  MoveC 7172 to (-6.47, 57.05, -11) mm, rotated rx -180 ry 0 rz 90 deg; joints [75.622, -17.705, 85.85, 0, 21.855, 75.622] to (-5.97, 56.82, -11) mm, rotated rx 180 ry 0 rz 90 deg; joints [75.618, -17.695, 85.811, 0, 21.884, 75.618]
  MoveC 7173 to (11.96, 58.42, -11) mm, rotated rx 180 ry 0 rz 90 deg; joints [75.821, -17.382, 84.57, 0, 22.812, 75.821] to (29.85, 60.38, -11) mm, rotated rx -180 ry 0 rz 90 deg; joints [76.031, -17.055, 83.319, 0, 23.736, 76.031]
  MoveC 7174 to (37.63, 61.41, -11) mm, rotated rx 180 ry 0 rz 90 deg; joints [76.126, -16.91, 82.773, 0, 24.137, 76.126] to (45.39, 62.55, -11) mm, rotated rx -180 ry 0 rz 90 deg; joints [76.225, -16.762, 82.226, 0, 24.537, 76.225]
  MoveL 7175 to (45.39, 69.07, -11) mm, rotated rx 180 ry 0 rz 90 deg; joints [76.435, -16.794, 82.342, 0, 24.452, 76.435]
  MoveC 7176 to (32.64, 69.9, -11) mm, rotated rx 180 ry 0 rz 90 deg; joints [76.362, -17.047, 83.287, 0, 23.76, 76.362] to (19.88, 70.48, -11) mm, rotated rx -180 ry 0 rz 90 deg; joints [76.279, -17.291, 84.218, 0, 23.073, 76.279]
  MoveC 7177 to (17, 70.58, -11) mm, rotated rx 180 ry 0 rz 90 deg; joints [76.26, -17.344, 84.426, 0, 22.919, 76.26] to (14.12, 70.67, -11) mm, rotated rx 180 ry 0 rz 90 deg; joints [76.24, -17.398, 84.633, 0, 22.765, 76.24]
  MoveL 7178 to (13.87, 63.13, -11) mm, rotated rx -180 ry 0 rz 90 deg; joints [75.991, -17.368, 84.518, 0, 22.85, 75.991]
  MoveL 7179 to (13.87, 63.13, -8) mm, rotated rx 180 ry 0 rz 90 deg; joints [75.991, -17.522, 84.62, 0, 22.902, 75.991]
  Establecer velocidad (1000.0 mm/s)
  MoveL 7180 to (13.87, 63.13, 10) mm, rotated rx 180 ry 0 rz 90 deg; joints [75.991, -18.443, 85.222, 0, 23.22, 75.991]
  Establecer velocidad (66.7 mm/s)
  MoveL 7181 to (-0.84, 59.62, 10) mm, rotated rx 180 ry 0 rz 90 deg; joints [75.754, -18.697, 86.204, 0, 22.493, 75.754]
  MoveL 7182 to (-0.84, 59.62, -8) mm, rotated rx -180 ry 0 rz 90 deg; joints [75.754, -17.772, 85.602, 0, 22.17, 75.754]
  MoveL 7183 to (0.35, 58.68, -8.41) mm, rotated rx -180 ry 0 rz 90 deg; joints [75.733, -17.725, 85.487, 0, 22.239, 75.733]
  MoveL 7184 to (1.74, 58.06, -8.81) mm, rotated rx 180 ry 0 rz 90 deg; joints [75.724, -17.677, 85.364, 0, 22.313, 75.724]
  MoveL 7185 to (3.23, 57.78, -9.22) mm, rotated rx -180 ry 0 rz 90 deg; joints [75.727, -17.628, 85.239, 0, 22.389, 75.727]
  MoveL 7186 to (4.75, 57.85, -9.62) mm, rotated rx -180 ry 0 rz 90 deg; joints [75.742, -17.58, 85.119, 0, 22.461, 75.742]
  MoveL 7187 to (6.21, 58.28, -10.03) mm, rotated rx 180 ry 0 rz 90 deg; joints [75.769, -17.535, 85.009, 0, 22.526, 75.769]
  MoveL 7188 to (7.53, 59.03, -10.44) mm, rotated rx 180 ry 0 rz 90 deg; joints [75.804, -17.494, 84.915, 0, 22.579, 75.804]
  MoveL 7189 to (8.65, 60.06, -10.84) mm, rotated rx 180 ry 0 rz 90 deg; joints [75.847, -17.458, 84.841, 0, 22.617, 75.847]
  MoveL 7190 to (9.46, 61.34, -11.25) mm, rotated rx 180 ry 0 rz 90 deg; joints [75.896, -17.428, 84.792, 0, 22.636, 75.896]
  MoveL 7191 to (14.11, 70.46, -11.25) mm, rotated rx 180 ry 0 rz 90 deg; joints [76.233, -17.384, 84.621, 0, 22.763, 76.233]
  MoveL 7192 to (7.11, 70.69, -11.25) mm, rotated rx 180 ry 0 rz 90 deg; joints [76.184, -17.512, 85.124, 0, 22.388, 76.184]
  MoveL 7193 to (-16.58, 71.34, -11.25) mm, rotated rx -180 ry 0 rz 90 deg; joints [76.011, -17.928, 86.802, 0, 21.125, 76.011]
  MoveC 7194 to (-18.77, 68.61, -11.25) mm, rotated rx 180 ry 0 rz 90 deg; joints [75.902, -17.953, 86.907, 0, 21.046, 75.902] to (-18.5, 65.12, -11.25) mm, rotated rx -180 ry 0 rz 90 deg; joints [75.788, -17.933, 86.827, 0, 21.107, 75.788]
  MoveL 7195 to (-8.05, 58.36, -11.25) mm, rotated rx 180 ry 0 rz 90 deg; joints [75.652, -17.726, 85.977, 0, 21.749, 75.652]
  MoveL 7196 to (-6.15, 57.11, -11.25) mm, rotated rx 180 ry 0 rz 90 deg; joints [75.626, -17.687, 85.82, 0, 21.867, 75.626]
  MoveC 7197 to (-5.87, 56.99, -11.25) mm, rotated rx -180 ry 0 rz 90 deg; joints [75.625, -17.681, 85.798, 0, 21.883, 75.625] to (-5.57, 56.96, -11.25) mm, rotated rx -180 ry 0 rz 90 deg; joints [75.627, -17.676, 85.777, 0, 21.899, 75.627]
  MoveC 7198 to (11.68, 58.54, -11.25) mm, rotated rx -180 ry 0 rz 90 deg; joints [75.823, -17.374, 84.583, 0, 22.791, 75.823] to (28.9, 60.45, -11.25) mm, rotated rx 180 ry 0 rz 90 deg; joints [76.025, -17.061, 83.381, 0, 23.681, 76.025]
  MoveL 7199 to (40.27, 62.01, -11.25) mm, rotated rx -180 ry 0 rz 90 deg; joints [76.167, -16.848, 82.582, 0, 24.266, 76.167]
  MoveL 7200 to (42.53, 62.35, -11.25) mm, rotated rx -180 ry 0 rz 90 deg; joints [76.196, -16.805, 82.423, 0, 24.382, 76.196]
  MoveL 7201 to (42.53, 69.03, -11.25) mm, rotated rx 180 ry 0 rz 90 deg; joints [76.411, -16.838, 82.542, 0, 24.295, 76.411]
  MoveC 7202 to (29.09, 69.85, -11.25) mm, rotated rx 180 ry 0 rz 90 deg; joints [76.332, -17.102, 83.534, 0, 23.567, 76.332] to (15.63, 70.41, -11.25) mm, rotated rx 180 ry 0 rz 90 deg; joints [76.243, -17.356, 84.512, 0, 22.844, 76.243]
  MoveL 7203 to (14.11, 70.46, -11.25) mm, rotated rx 180 ry 0 rz 90 deg; joints [76.233, -17.384, 84.621, 0, 22.763, 76.233]
  MoveL 7204 to (13.87, 62.91, -11.25) mm, rotated rx 180 ry 0 rz 90 deg; joints [75.984, -17.354, 84.506, 0, 22.849, 75.984]
  MoveL 7205 to (13.87, 62.91, -8.25) mm, rotated rx 180 ry 0 rz 90 deg; joints [75.984, -17.508, 84.608, 0, 22.9, 75.984]
  Establecer velocidad (1000.0 mm/s)
  MoveL 7206 to (13.87, 62.91, 10) mm, rotated rx -180 ry 0 rz 90 deg; joints [75.984, -18.442, 85.219, 0, 23.223, 75.984]
  Establecer velocidad (66.7 mm/s)
  MoveL 7207 to (34.75, 17.39, 10) mm, rotated rx 180 ry 0 rz 90 deg; joints [74.689, -17.806, 82.854, 0, 24.952, 74.689]
  MoveL 7208 to (34.75, 17.39, -8) mm, rotated rx 180 ry 0 rz 90 deg; joints [74.689, -16.893, 82.249, 0, 24.644, 74.689]
  MoveL 7209 to (34.95, 18.89, -8.41) mm, rotated rx 180 ry 0 rz 90 deg; joints [74.738, -16.877, 82.251, 0, 24.626, 74.738]
  MoveL 7210 to (34.77, 20.4, -8.81) mm, rotated rx -180 ry 0 rz 90 deg; joints [74.785, -16.868, 82.28, 0, 24.588, 74.785]
  MoveL 7211 to (34.27, 21.84, -9.22) mm, rotated rx 180 ry 0 rz 90 deg; joints [74.827, -16.865, 82.332, 0, 24.534, 74.827]
  MoveL 7212 to (33.46, 23.12, -9.62) mm, rotated rx -180 ry 0 rz 90 deg; joints [74.861, -16.867, 82.402, 0, 24.465, 74.861]
  MoveL 7213 to (32.38, 24.2, -10.03) mm, rotated rx 180 ry 0 rz 90 deg; joints [74.886, -16.874, 82.488, 0, 24.386, 74.886]
  MoveL 7214 to (31.1, 25.01, -10.44) mm, rotated rx -180 ry 0 rz 90 deg; joints [74.901, -16.882, 82.583, 0, 24.299, 74.901]
  MoveL 7215 to (29.66, 25.51, -10.84) mm, rotated rx 180 ry 0 rz 90 deg; joints [74.904, -16.892, 82.683, 0, 24.209, 74.904]
  MoveL 7216 to (28.15, 25.66, -11.25) mm, rotated rx -180 ry 0 rz 90 deg; joints [74.896, -16.902, 82.781, 0, 24.12, 74.896]
  MoveC 7217 to (21.42, 25.67, -11.25) mm, rotated rx 180 ry 0 rz 90 deg; joints [74.838, -17.031, 83.268, 0, 23.763, 74.838] to (14.69, 25.64, -11.25) mm, rotated rx 180 ry 0 rz 90 deg; joints [74.778, -17.159, 83.751, 0, 23.408, 74.778]
  MoveL 7218 to (13.74, 25.57, -11.25) mm, rotated rx 180 ry 0 rz 90 deg; joints [74.767, -17.176, 83.818, 0, 23.358, 74.767]
  MoveC 7219 to (11.74, 24.17, -11.25) mm, rotated rx 180 ry 0 rz 90 deg; joints [74.704, -17.206, 83.934, 0, 23.273, 74.704] to (11.18, 21.8, -11.25) mm, rotated rx 180 ry 0 rz 90 deg; joints [74.622, -17.205, 83.927, 0, 23.277, 74.622]
  MoveL 7220 to (11.34, 21.32, -11.25) mm, rotated rx 180 ry 0 rz 90 deg; joints [74.609, -17.199, 83.906, 0, 23.293, 74.609]
  MoveL 7221 to (14.96, 11.54, -11.25) mm, rotated rx 180 ry 0 rz 90 deg; joints [74.325, -17.08, 83.453, 0, 23.628, 74.325]
  MoveC 7222 to (15.41, 10.71, -11.25) mm, rotated rx 180 ry 0 rz 90 deg; joints [74.303, -17.067, 83.403, 0, 23.664, 74.303] to (16.08, 10.04, -11.25) mm, rotated rx 180 ry 0 rz 90 deg; joints [74.287, -17.051, 83.342, 0, 23.709, 74.287]
  MoveL 7223 to (27.98, 1.22, -11.25) mm, rotated rx -180 ry 0 rz 90 deg; joints [74.113, -16.773, 82.303, 0, 24.47, 74.113]
  MoveC 7224 to (28.43, 0.91, -11.25) mm, rotated rx 180 ry 0 rz 90 deg; joints [74.107, -16.762, 82.264, 0, 24.498, 74.107] to (28.9, 0.64, -11.25) mm, rotated rx -180 ry 0 rz 90 deg; joints [74.102, -16.751, 82.224, 0, 24.528, 74.102]
  MoveC 7225 to (31.23, 0.68, -11.25) mm, rotated rx 180 ry 0 rz 90 deg; joints [74.125, -16.706, 82.055, 0, 24.65, 74.125] to (33.09, 2.08, -11.25) mm, rotated rx 180 ry 0 rz 90 deg; joints [74.186, -16.677, 81.949, 0, 24.728, 74.186]
  MoveL 7226 to (33.64, 2.87, -11.25) mm, rotated rx 180 ry 0 rz 90 deg; joints [74.216, -16.67, 81.925, 0, 24.745, 74.216]
  MoveL 7227 to (42.53, 15.9, -11.25) mm, rotated rx 180 ry 0 rz 90 deg; joints [74.709, -16.565, 81.54, 0, 25.025, 74.709]
  MoveL 7228 to (42.53, 25.35, -11.25) mm, rotated rx -180 ry 0 rz 90 deg; joints [75.01, -16.616, 81.727, 0, 24.889, 75.01]
  MoveL 7229 to (42.3, 25.48, -11.25) mm, rotated rx -180 ry 0 rz 90 deg; joints [75.012, -16.621, 81.747, 0, 24.875, 75.012]
  MoveL 7230 to (41.22, 25.52, -11.25) mm, rotated rx 180 ry 0 rz 90 deg; joints [75.004, -16.643, 81.827, 0, 24.817, 75.004]
  MoveC 7231 to (34.69, 25.61, -11.25) mm, rotated rx -180 ry 0 rz 90 deg; joints [74.951, -16.774, 82.306, 0, 24.468, 74.951] to (28.15, 25.66, -11.25) mm, rotated rx -180 ry 0 rz 90 deg; joints [74.896, -16.902, 82.781, 0, 24.12, 74.896]
  MoveL 7232 to (28.12, 18.11, -11.25) mm, rotated rx -180 ry 0 rz 90 deg; joints [74.654, -16.863, 82.635, 0, 24.228, 74.654]
  MoveL 7233 to (28.12, 18.11, -8.25) mm, rotated rx -180 ry 0 rz 90 deg; joints [74.654, -17.015, 82.737, 0, 24.278, 74.654]
  Establecer velocidad (1000.0 mm/s)
  MoveL 7234 to (28.12, 18.11, 10) mm, rotated rx 180 ry 0 rz 90 deg; joints [74.654, -17.942, 83.35, 0, 24.592, 74.654]
  Establecer velocidad (66.7 mm/s)
  MoveL 7235 to (14.48, -62.46, 10) mm, rotated rx 180 ry 0 rz 90 deg; joints [71.966, -17.733, 82.59, 0, 25.143, 71.966]
  MoveL 7236 to (14.48, -62.46, -8) mm, rotated rx -180 ry 0 rz 90 deg; joints [71.966, -16.821, 81.985, 0, 24.836, 71.966]
  MoveL 7237 to (14.35, -63.97, -8.41) mm, rotated rx 180 ry 0 rz 90 deg; joints [71.918, -16.793, 81.945, 0, 24.848, 71.918]
  MoveL 7238 to (14.59, -65.48, -8.81) mm, rotated rx 180 ry 0 rz 90 deg; joints [71.873, -16.758, 81.878, 0, 24.88, 71.873]
  MoveL 7239 to (15.16, -66.89, -9.22) mm, rotated rx 180 ry 0 rz 90 deg; joints [71.835, -16.717, 81.79, 0, 24.927, 71.835]
  MoveL 7240 to (16.03, -68.13, -9.62) mm, rotated rx -180 ry 0 rz 90 deg; joints [71.804, -16.671, 81.684, 0, 24.987, 71.804]
  MoveL 7241 to (17.15, -69.16, -10.03) mm, rotated rx 180 ry 0 rz 90 deg; joints [71.784, -16.622, 81.565, 0, 25.057, 71.784]
  MoveL 7242 to (18.47, -69.91, -10.44) mm, rotated rx 180 ry 0 rz 90 deg; joints [71.774, -16.57, 81.438, 0, 25.132, 71.774]
  MoveL 7243 to (19.92, -70.36, -10.84) mm, rotated rx 180 ry 0 rz 90 deg; joints [71.775, -16.517, 81.308, 0, 25.209, 71.775]
  MoveL 7244 to (21.44, -70.43, -11.25) mm, rotated rx 180 ry 0 rz 90 deg; joints [71.788, -16.466, 81.182, 0, 25.284, 71.788]
  MoveC 7245 to (30.97, -70.02, -11.25) mm, rotated rx 180 ry 0 rz 90 deg; joints [71.898, -16.275, 80.498, 0, 25.777, 71.898] to (40.49, -69.51, -11.25) mm, rotated rx -180 ry 0 rz 90 deg; joints [72.01, -16.08, 79.81, 0, 26.27, 72.01]
  MoveC 7246 to (41.74, -68.34, -11.25) mm, rotated rx -180 ry 0 rz 90 deg; joints [72.059, -16.062, 79.746, 0, 26.316, 72.059] to (42.53, -66.81, -11.25) mm, rotated rx -180 ry 0 rz 90 deg; joints [72.114, -16.055, 79.723, 0, 26.332, 72.114]
  MoveL 7247 to (42.53, -62.79, -11.25) mm, rotated rx -180 ry 0 rz 90 deg; joints [72.239, -16.082, 79.819, 0, 26.263, 72.239]
  MoveC 7248 to (32.93, -50.94, -11.25) mm, rotated rx 180 ry 0 rz 90 deg; joints [72.513, -16.36, 80.802, 0, 25.558, 72.513] to (23.22, -39.19, -11.25) mm, rotated rx -180 ry 0 rz 90 deg; joints [72.786, -16.63, 81.777, 0, 24.853, 72.786]
  MoveL 7249 to (22.31, -38.38, -11.25) mm, rotated rx 180 ry 0 rz 90 deg; joints [72.803, -16.653, 81.861, 0, 24.792, 72.803]
  MoveL 7250 to (13.74, -31.32, -11.25) mm, rotated rx 180 ry 0 rz 90 deg; joints [72.943, -16.863, 82.636, 0, 24.227, 72.943]
  MoveC 7251 to (11.26, -30.82, -11.25) mm, rotated rx 180 ry 0 rz 90 deg; joints [72.935, -16.914, 82.826, 0, 24.088, 72.935] to (9, -31.97, -11.25) mm, rotated rx 180 ry 0 rz 90 deg; joints [72.876, -16.95, 82.962, 0, 23.988, 72.876]
  MoveC 7252 to (8.77, -32.34, -11.25) mm, rotated rx -180 ry 0 rz 90 deg; joints [72.862, -16.952, 82.971, 0, 23.982, 72.862] to (8.61, -32.74, -11.25) mm, rotated rx -180 ry 0 rz 90 deg; joints [72.848, -16.953, 82.973, 0, 23.98, 72.848]
  MoveL 7253 to (-0.76, -67.29, -11.25) mm, rotated rx 180 ry 0 rz 90 deg; joints [71.657, -16.921, 82.853, 0, 24.068, 71.657]
  MoveC 7254 to (-0.84, -67.76, -11.25) mm, rotated rx -180 ry 0 rz 90 deg; joints [71.641, -16.919, 82.847, 0, 24.072, 71.641] to (-0.81, -68.23, -11.25) mm, rotated rx 180 ry 0 rz 90 deg; joints [71.626, -16.916, 82.833, 0, 24.082, 71.626]
  MoveC 7255 to (0.29, -70.18, -11.25) mm, rotated rx 180 ry 0 rz 90 deg; joints [71.576, -16.882, 82.709, 0, 24.173, 71.576] to (2.37, -71.02, -11.25) mm, rotated rx -180 ry 0 rz 90 deg; joints [71.572, -16.837, 82.541, 0, 24.296, 71.572]
  MoveC 7256 to (11.91, -70.77, -11.25) mm, rotated rx -180 ry 0 rz 90 deg; joints [71.679, -16.653, 81.863, 0, 24.79, 71.679] to (21.44, -70.43, -11.25) mm, rotated rx 180 ry 0 rz 90 deg; joints [71.788, -16.466, 81.182, 0, 25.284, 71.788]
  MoveL 7257 to (21.14, -62.89, -11.25) mm, rotated rx 180 ry 0 rz 90 deg; joints [72.021, -16.521, 81.383, 0, 25.138, 72.021]
  MoveL 7258 to (21.14, -62.89, -8.25) mm, rotated rx 180 ry 0 rz 90 deg; joints [72.021, -16.673, 81.485, 0, 25.188, 72.021]
  Establecer velocidad (1000.0 mm/s)
  MoveL 7259 to (21.14, -62.89, 10) mm, rotated rx 180 ry 0 rz 90 deg; joints [72.021, -17.596, 82.099, 0, 25.497, 72.021]
  Establecer velocidad (66.7 mm/s)
  MoveL 7260 to (-37.75, -51.92, 10) mm, rotated rx 180 ry 0 rz 90 deg; joints [71.757, -18.775, 86.512, 0, 22.263, 71.757]
  MoveL 7261 to (-37.75, -51.92, -8) mm, rotated rx 180 ry 0 rz 90 deg; joints [71.757, -17.849, 85.91, 0, 21.939, 71.757]
  MoveL 7262 to (-36.33, -52.48, -8.41) mm, rotated rx -180 ry 0 rz 90 deg; joints [71.754, -17.801, 85.786, 0, 22.015, 71.754]
  MoveL 7263 to (-34.83, -52.68, -8.81) mm, rotated rx 180 ry 0 rz 90 deg; joints [71.764, -17.753, 85.664, 0, 22.089, 71.764]
  MoveL 7264 to (-33.31, -52.54, -9.22) mm, rotated rx 180 ry 0 rz 90 deg; joints [71.784, -17.706, 85.548, 0, 22.158, 71.784]
  MoveL 7265 to (-31.87, -52.07, -9.62) mm, rotated rx 180 ry 0 rz 90 deg; joints [71.815, -17.663, 85.445, 0, 22.218, 71.815]
  MoveL 7266 to (-30.56, -51.29, -10.03) mm, rotated rx -180 ry 0 rz 90 deg; joints [71.854, -17.624, 85.358, 0, 22.265, 71.854]
  MoveL 7267 to (-29.46, -50.25, -10.44) mm, rotated rx 180 ry 0 rz 90 deg; joints [71.899, -17.589, 85.292, 0, 22.297, 71.899]
  MoveL 7268 to (-28.62, -48.98, -10.84) mm, rotated rx 180 ry 0 rz 90 deg; joints [71.949, -17.561, 85.248, 0, 22.313, 71.949]
  MoveL 7269 to (-28.11, -47.55, -11.25) mm, rotated rx -180 ry 0 rz 90 deg; joints [72, -17.539, 85.231, 0, 22.308, 72]
  MoveL 7270 to (-22.44, -25.59, -11.25) mm, rotated rx 180 ry 0 rz 90 deg; joints [72.769, -17.562, 85.322, 0, 22.24, 72.769]
  MoveC 7271 to (-22.4, -25.35, -11.25) mm, rotated rx 180 ry 0 rz 90 deg; joints [72.777, -17.563, 85.324, 0, 22.238, 72.777] to (-22.41, -25.11, -11.25) mm, rotated rx 180 ry 0 rz 90 deg; joints [72.784, -17.564, 85.33, 0, 22.234, 72.784]
  MoveC 7272 to (-23.45, -22.93, -11.25) mm, rotated rx 180 ry 0 rz 90 deg; joints [72.845, -17.594, 85.45, 0, 22.145, 72.845] to (-25.59, -21.78, -11.25) mm, rotated rx -180 ry 0 rz 90 deg; joints [72.861, -17.638, 85.623, 0, 22.015, 72.861]
  MoveL 7273 to (-26.06, -21.85, -11.25) mm, rotated rx -180 ry 0 rz 90 deg; joints [72.854, -17.646, 85.654, 0, 21.991, 72.854]
  MoveL 7274 to (-33.64, -23.38, -11.25) mm, rotated rx -180 ry 0 rz 90 deg; joints [72.727, -17.768, 86.147, 0, 21.621, 72.727]
  MoveL 7275 to (-63.02, -29.41, -11.25) mm, rotated rx 180 ry 0 rz 90 deg; joints [72.225, -18.217, 88.022, 0, 20.195, 72.225]
  MoveL 7276 to (-70.18, -30.91, -11.25) mm, rotated rx 180 ry 0 rz 90 deg; joints [72.099, -18.321, 88.472, 0, 19.849, 72.099]
  MoveC 7277 to (-71.74, -31.8, -11.25) mm, rotated rx 180 ry 0 rz 90 deg; joints [72.052, -18.341, 88.557, 0, 19.783, 72.052] to (-72.48, -33.43, -11.25) mm, rotated rx -180 ry 0 rz 90 deg; joints [71.99, -18.344, 88.572, 0, 19.772, 71.99]
  MoveL 7278 to (-72.5, -33.64, -11.25) mm, rotated rx 180 ry 0 rz 90 deg; joints [71.983, -18.343, 88.569, 0, 19.775, 71.983]
  MoveL 7279 to (-72.51, -68.7, -11.25) mm, rotated rx 180 ry 0 rz 90 deg; joints [70.828, -18.16, 87.778, 0, 20.382, 70.828]
  MoveL 7280 to (-72.5, -69.19, -11.25) mm, rotated rx 180 ry 0 rz 90 deg; joints [70.812, -18.157, 87.766, 0, 20.391, 70.812]
  MoveC 7281 to (-71.63, -71.22, -11.25) mm, rotated rx 180 ry 0 rz 90 deg; joints [70.756, -18.132, 87.66, 0, 20.472, 70.756] to (-69.61, -72.07, -11.25) mm, rotated rx -180 ry 0 rz 90 deg; joints [70.751, -18.095, 87.504, 0, 20.592, 70.751]
  MoveL 7282 to (-68.7, -72.08, -11.25) mm, rotated rx 180 ry 0 rz 90 deg; joints [70.761, -18.081, 87.443, 0, 20.638, 70.761]
  MoveL 7283 to (-62.07, -72, -11.25) mm, rotated rx 180 ry 0 rz 90 deg; joints [70.839, -17.974, 86.997, 0, 20.978, 70.839]
  MoveL 7284 to (-60.18, -71.98, -11.25) mm, rotated rx 180 ry 0 rz 90 deg; joints [70.861, -17.944, 86.869, 0, 21.075, 70.861]
  MoveL 7285 to (-37.43, -71.64, -11.25) mm, rotated rx 180 ry 0 rz 90 deg; joints [71.125, -17.562, 85.321, 0, 22.241, 71.125]
  MoveL 7286 to (-36.53, -71.61, -11.25) mm, rotated rx -180 ry 0 rz 90 deg; joints [71.135, -17.546, 85.259, 0, 22.287, 71.135]
  MoveC 7287 to (-34.82, -71, -11.25) mm, rotated rx 180 ry 0 rz 90 deg; joints [71.174, -17.52, 85.155, 0, 22.365, 71.174] to (-33.8, -69.51, -11.25) mm, rotated rx -180 ry 0 rz 90 deg; joints [71.233, -17.511, 85.12, 0, 22.391, 71.233]
  MoveL 7288 to (-33.64, -68.97, -11.25) mm, rotated rx -180 ry 0 rz 90 deg; joints [71.252, -17.512, 85.121, 0, 22.39, 71.252]
  MoveL 7289 to (-32.83, -65.86, -11.25) mm, rotated rx -180 ry 0 rz 90 deg; joints [71.36, -17.516, 85.138, 0, 22.378, 71.36]
  MoveL 7290 to (-28.11, -47.55, -11.25) mm, rotated rx -180 ry 0 rz 90 deg; joints [72, -17.539, 85.231, 0, 22.308, 72]
  MoveL 7291 to (-35.42, -45.67, -11.25) mm, rotated rx 180 ry 0 rz 90 deg; joints [71.984, -17.677, 85.78, 0, 21.897, 71.984]
  MoveL 7292 to (-35.42, -45.67, -8.25) mm, rotated rx -180 ry 0 rz 90 deg; joints [71.984, -17.831, 85.882, 0, 21.949, 71.984]
  Establecer velocidad (1000.0 mm/s)
  MoveL 7293 to (-35.42, -45.67, 10) mm, rotated rx -180 ry 0 rz 90 deg; joints [71.984, -18.77, 86.493, 0, 22.277, 71.984]
  Establecer velocidad (66.7 mm/s)
  MoveL 7294 to (-64.27, 35.76, 10) mm, rotated rx 180 ry 0 rz 90 deg; joints [74.392, -19.648, 90.137, 0, 19.51, 74.392]
  MoveL 7295 to (-64.27, 35.76, -8) mm, rotated rx 180 ry 0 rz 90 deg; joints [74.392, -18.706, 89.535, 0, 19.172, 74.392]
  MoveL 7296 to (-65.78, 35.94, -8.41) mm, rotated rx -180 ry 0 rz 90 deg; joints [74.384, -18.709, 89.626, 0, 19.083, 74.384]
  MoveL 7297 to (-67.28, 35.76, -8.81) mm, rotated rx 180 ry 0 rz 90 deg; joints [74.364, -18.709, 89.71, 0, 18.999, 74.364]
  MoveL 7298 to (-68.71, 35.25, -9.22) mm, rotated rx -180 ry 0 rz 90 deg; joints [74.333, -18.707, 89.782, 0, 18.925, 74.333]
  MoveL 7299 to (-70, 34.43, -9.62) mm, rotated rx -180 ry 0 rz 90 deg; joints [74.293, -18.701, 89.839, 0, 18.862, 74.293]
  MoveL 7300 to (-71.07, 33.35, -10.03) mm, rotated rx -180 ry 0 rz 90 deg; joints [74.246, -18.691, 89.876, 0, 18.815, 74.246]
  MoveL 7301 to (-71.87, 32.06, -10.44) mm, rotated rx 180 ry 0 rz 90 deg; joints [74.195, -18.676, 89.892, 0, 18.784, 74.195]
  MoveL 7302 to (-72.37, 30.63, -10.84) mm, rotated rx -180 ry 0 rz 90 deg; joints [74.141, -18.656, 89.884, 0, 18.772, 74.141]
  MoveL 7303 to (-72.51, 29.12, -11.25) mm, rotated rx 180 ry 0 rz 90 deg; joints [74.089, -18.631, 89.851, 0, 18.78, 74.089]
  MoveL 7304 to (-72.51, 3.32, -11.25) mm, rotated rx -180 ry 0 rz 90 deg; joints [73.217, -18.519, 89.345, 0, 19.174, 73.217]
  MoveL 7305 to (-72.49, 2.64, -11.25) mm, rotated rx -180 ry 0 rz 90 deg; joints [73.195, -18.515, 89.33, 0, 19.185, 73.195]
  MoveC 7306 to (-71.39, 0.6, -11.25) mm, rotated rx 180 ry 0 rz 90 deg; joints [73.137, -18.49, 89.215, 0, 19.275, 73.137] to (-69.18, -0.09, -11.25) mm, rotated rx -180 ry 0 rz 90 deg; joints [73.137, -18.453, 89.053, 0, 19.401, 73.137]
  MoveC 7307 to (-46.42, 5.25, -11.25) mm, rotated rx -180 ry 0 rz 90 deg; joints [73.542, -18.123, 87.62, 0, 20.502, 73.542] to (-23.69, 10.68, -11.25) mm, rotated rx -180 ry 0 rz 90 deg; joints [73.94, -17.772, 86.163, 0, 21.608, 73.94]
  MoveC 7308 to (-23.01, 10.94, -11.25) mm, rotated rx 180 ry 0 rz 90 deg; joints [73.955, -17.761, 86.122, 0, 21.64, 73.955] to (-22.43, 11.37, -11.25) mm, rotated rx -180 ry 0 rz 90 deg; joints [73.975, -17.754, 86.09, 0, 21.663, 73.975]
  MoveC 7309 to (-21.58, 12.67, -11.25) mm, rotated rx 180 ry 0 rz 90 deg; joints [74.025, -17.745, 86.056, 0, 21.689, 74.025] to (-21.36, 14.21, -11.25) mm, rotated rx 180 ry 0 rz 90 deg; joints [74.078, -17.749, 86.072, 0, 21.677, 74.078]
  MoveC 7310 to (-21.48, 14.65, -11.25) mm, rotated rx -180 ry 0 rz 90 deg; joints [74.091, -17.753, 86.089, 0, 21.664, 74.091] to (-21.62, 15.09, -11.25) mm, rotated rx -180 ry 0 rz 90 deg; joints [74.104, -17.758, 86.107, 0, 21.651, 74.104]
  MoveL 7311 to (-27.11, 30.54, -11.25) mm, rotated rx -180 ry 0 rz 90 deg; joints [74.563, -17.924, 86.789, 0, 21.135, 74.563]
  MoveC 7312 to (-27.43, 31.26, -11.25) mm, rotated rx -180 ry 0 rz 90 deg; joints [74.584, -17.933, 86.825, 0, 21.108, 74.584] to (-27.87, 31.91, -11.25) mm, rotated rx 180 ry 0 rz 90 deg; joints [74.602, -17.943, 86.868, 0, 21.075, 74.602]
  MoveL 7313 to (-27.96, 31.99, -11.25) mm, rotated rx 180 ry 0 rz 90 deg; joints [74.604, -17.945, 86.876, 0, 21.07, 74.604]
  MoveL 7314 to (-28.9, 32.69, -11.25) mm, rotated rx 180 ry 0 rz 90 deg; joints [74.618, -17.964, 86.954, 0, 21.01, 74.618]
  MoveC 7315 to (-48.55, 45.47, -11.25) mm, rotated rx 180 ry 0 rz 90 deg; joints [74.866, -18.337, 88.541, 0, 19.796, 74.866] to (-68.23, 58.2, -11.25) mm, rotated rx -180 ry 0 rz 90 deg; joints [75.119, -18.685, 90.101, 0, 18.584, 75.119]
  MoveC 7316 to (-70.59, 58.01, -11.25) mm, rotated rx -180 ry 0 rz 90 deg; joints [75.091, -18.719, 90.255, 0, 18.463, 75.091] to (-72.31, 56.4, -11.25) mm, rotated rx 180 ry 0 rz 90 deg; joints [75.02, -18.737, 90.342, 0, 18.396, 75.02]
  MoveC 7317 to (-72.46, 56.01, -11.25) mm, rotated rx 180 ry 0 rz 90 deg; joints [75.005, -18.738, 90.345, 0, 18.393, 75.005] to (-72.51, 55.6, -11.25) mm, rotated rx -180 ry 0 rz 90 deg; joints [74.991, -18.737, 90.341, 0, 18.396, 74.991]
  MoveL 7318 to (-72.51, 29.12, -11.25) mm, rotated rx 180 ry 0 rz 90 deg; joints [74.089, -18.631, 89.851, 0, 18.78, 74.089]
  MoveL 7319 to (-64.96, 29.12, -11.25) mm, rotated rx 180 ry 0 rz 90 deg; joints [74.161, -18.519, 89.345, 0, 19.174, 74.161]
  MoveL 7320 to (-64.96, 29.12, -8.25) mm, rotated rx 180 ry 0 rz 90 deg; joints [74.161, -18.676, 89.447, 0, 19.229, 74.161]
  Establecer velocidad (1000.0 mm/s)
  MoveL 7321 to (-64.96, 29.12, 10) mm, rotated rx 180 ry 0 rz 90 deg; joints [74.161, -19.63, 90.058, 0, 19.572, 74.161]
  Establecer velocidad (66.7 mm/s)
  MoveL 7322 to (-64.1, 35.76, 10) mm, rotated rx 180 ry 0 rz 90 deg; joints [74.394, -19.645, 90.126, 0, 19.519, 74.394]
  MoveL 7323 to (-64.1, 35.76, -8.25) mm, rotated rx -180 ry 0 rz 90 deg; joints [74.394, -18.691, 89.515, 0, 19.176, 74.394]
  MoveL 7324 to (-65.61, 35.94, -8.66) mm, rotated rx 180 ry 0 rz 90 deg; joints [74.386, -18.693, 89.606, 0, 19.087, 74.386]
  MoveL 7325 to (-67.12, 35.76, -9.06) mm, rotated rx 180 ry 0 rz 90 deg; joints [74.366, -18.693, 89.69, 0, 19.003, 74.366]
  MoveL 7326 to (-68.55, 35.25, -9.47) mm, rotated rx 180 ry 0 rz 90 deg; joints [74.335, -18.691, 89.763, 0, 18.929, 74.335]
  MoveL 7327 to (-69.83, 34.43, -9.88) mm, rotated rx 180 ry 0 rz 90 deg; joints [74.295, -18.686, 89.819, 0, 18.866, 74.295]
  MoveL 7328 to (-70.9, 33.35, -10.28) mm, rotated rx -180 ry 0 rz 90 deg; joints [74.248, -18.675, 89.857, 0, 18.819, 74.248]
  MoveL 7329 to (-71.71, 32.06, -10.69) mm, rotated rx -180 ry 0 rz 90 deg; joints [74.196, -18.661, 89.872, 0, 18.788, 74.196]
  MoveL 7330 to (-72.2, 30.63, -11.09) mm, rotated rx 180 ry 0 rz 90 deg; joints [74.143, -18.641, 89.865, 0, 18.776, 74.143]
  MoveL 7331 to (-72.34, 29.12, -11.5) mm, rotated rx -180 ry 0 rz 90 deg; joints [74.09, -18.615, 89.831, 0, 18.784, 74.09]
  MoveL 7332 to (-72.34, 3.32, -11.5) mm, rotated rx -180 ry 0 rz 90 deg; joints [73.219, -18.503, 89.325, 0, 19.178, 73.219]
  MoveL 7333 to (-72.34, 2.84, -11.5) mm, rotated rx 180 ry 0 rz 90 deg; joints [73.203, -18.501, 89.315, 0, 19.186, 73.203]
  MoveC 7334 to (-71.31, 0.83, -11.5) mm, rotated rx 180 ry 0 rz 90 deg; joints [73.146, -18.476, 89.206, 0, 19.271, 73.146] to (-69.18, 0.06, -11.5) mm, rotated rx 180 ry 0 rz 90 deg; joints [73.142, -18.441, 89.047, 0, 19.394, 73.142]
  MoveL 7335 to (-68.7, 0.15, -11.5) mm, rotated rx -180 ry 0 rz 90 deg; joints [73.15, -18.434, 89.017, 0, 19.417, 73.15]
  MoveL 7336 to (-44.07, 5.96, -11.5) mm, rotated rx -180 ry 0 rz 90 deg; joints [73.589, -18.075, 87.465, 0, 20.61, 73.589]
  MoveL 7337 to (-40.27, 6.88, -11.5) mm, rotated rx 180 ry 0 rz 90 deg; joints [73.656, -18.018, 87.224, 0, 20.794, 73.656]
  MoveL 7338 to (-24.17, 10.74, -11.5) mm, rotated rx 180 ry 0 rz 90 deg; joints [73.938, -17.767, 86.189, 0, 21.578, 73.938]
  MoveL 7339 to (-23.58, 10.9, -11.5) mm, rotated rx 180 ry 0 rz 90 deg; joints [73.948, -17.758, 86.152, 0, 21.606, 73.948]
  MoveC 7340 to (-21.92, 12.44, -11.5) mm, rotated rx -180 ry 0 rz 90 deg; joints [74.015, -17.737, 86.067, 0, 21.67, 74.015] to (-21.66, 14.69, -11.5) mm, rotated rx 180 ry 0 rz 90 deg; joints [74.091, -17.744, 86.094, 0, 21.65, 74.091]
  MoveL 7341 to (-21.98, 15.64, -11.5) mm, rotated rx 180 ry 0 rz 90 deg; joints [74.119, -17.754, 86.135, 0, 21.619, 74.119]
  MoveL 7342 to (-27.23, 30.43, -11.5) mm, rotated rx 180 ry 0 rz 90 deg; joints [74.559, -17.913, 86.787, 0, 21.126, 74.559]
  MoveC 7343 to (-27.54, 31.12, -11.5) mm, rotated rx 180 ry 0 rz 90 deg; joints [74.579, -17.921, 86.822, 0, 21.1, 74.579] to (-27.96, 31.76, -11.5) mm, rotated rx -180 ry 0 rz 90 deg; joints [74.596, -17.931, 86.863, 0, 21.068, 74.596]
  MoveC 7344 to (-28.45, 32.17, -11.5) mm, rotated rx -180 ry 0 rz 90 deg; joints [74.605, -17.941, 86.904, 0, 21.037, 74.605] to (-28.97, 32.53, -11.5) mm, rotated rx 180 ry 0 rz 90 deg; joints [74.612, -17.952, 86.947, 0, 21.004, 74.612]
  MoveC 7345 to (-48.53, 45.29, -11.5) mm, rotated rx -180 ry 0 rz 90 deg; joints [74.86, -18.323, 88.528, 0, 19.795, 74.86] to (-68.14, 57.98, -11.5) mm, rotated rx 180 ry 0 rz 90 deg; joints [75.112, -18.67, 90.082, 0, 18.588, 75.112]
  MoveC 7346 to (-70.35, 57.8, -11.5) mm, rotated rx -180 ry 0 rz 90 deg; joints [75.086, -18.701, 90.227, 0, 18.474, 75.086] to (-72.05, 56.38, -11.5) mm, rotated rx 180 ry 0 rz 90 deg; joints [75.022, -18.72, 90.315, 0, 18.405, 75.022]
  MoveC 7347 to (-72.27, 55.88, -11.5) mm, rotated rx -180 ry 0 rz 90 deg; joints [75.003, -18.721, 90.321, 0, 18.4, 75.003] to (-72.34, 55.35, -11.5) mm, rotated rx -180 ry 0 rz 90 deg; joints [74.984, -18.721, 90.317, 0, 18.404, 74.984]
  MoveL 7348 to (-72.34, 29.12, -11.5) mm, rotated rx -180 ry 0 rz 90 deg; joints [74.09, -18.615, 89.831, 0, 18.784, 74.09]
  MoveL 7349 to (-64.8, 29.12, -11.5) mm, rotated rx -180 ry 0 rz 90 deg; joints [74.163, -18.503, 89.325, 0, 19.178, 74.163]
  MoveL 7350 to (-64.8, 29.12, -8.5) mm, rotated rx 180 ry 0 rz 90 deg; joints [74.163, -18.66, 89.427, 0, 19.233, 74.163]
  Establecer velocidad (1000.0 mm/s)
  MoveL 7351 to (-64.8, 29.12, 10) mm, rotated rx 180 ry 0 rz 90 deg; joints [74.163, -19.627, 90.047, 0, 19.58, 74.163]
  Establecer velocidad (66.7 mm/s)
  MoveL 7352 to (-3.92, 59.74, 10) mm, rotated rx 180 ry 0 rz 90 deg; joints [75.732, -18.753, 86.424, 0, 22.329, 75.732]
  MoveL 7353 to (-3.92, 59.74, -8.25) mm, rotated rx -180 ry 0 rz 90 deg; joints [75.732, -17.814, 85.813, 0, 22.001, 75.732]
  MoveL 7354 to (-2.79, 58.73, -8.66) mm, rotated rx 180 ry 0 rz 90 deg; joints [75.708, -17.769, 85.701, 0, 22.067, 75.708]
  MoveL 7355 to (-1.43, 58.04, -9.06) mm, rotated rx 180 ry 0 rz 90 deg; joints [75.697, -17.721, 85.579, 0, 22.141, 75.697]
  MoveL 7356 to (0.04, 57.69, -9.47) mm, rotated rx -180 ry 0 rz 90 deg; joints [75.698, -17.672, 85.455, 0, 22.217, 75.698]
  MoveL 7357 to (1.56, 57.68, -9.88) mm, rotated rx 180 ry 0 rz 90 deg; joints [75.71, -17.624, 85.334, 0, 22.29, 75.71]
  MoveL 7358 to (3.04, 58.03, -10.28) mm, rotated rx 180 ry 0 rz 90 deg; joints [75.734, -17.578, 85.221, 0, 22.357, 75.734]
  MoveL 7359 to (4.4, 58.71, -10.69) mm, rotated rx 180 ry 0 rz 90 deg; joints [75.768, -17.536, 85.123, 0, 22.413, 75.768]
  MoveL 7360 to (5.57, 59.68, -11.09) mm, rotated rx 180 ry 0 rz 90 deg; joints [75.809, -17.499, 85.044, 0, 22.454, 75.809]
  MoveL 7361 to (6.45, 60.92, -11.5) mm, rotated rx 180 ry 0 rz 90 deg; joints [75.857, -17.467, 84.99, 0, 22.478, 75.857]
  MoveL 7362 to (11.88, 70.32, -11.5) mm, rotated rx 180 ry 0 rz 90 deg; joints [76.21, -17.411, 84.77, 0, 22.642, 76.21]
  MoveL 7363 to (9.95, 70.39, -11.5) mm, rotated rx 180 ry 0 rz 90 deg; joints [76.197, -17.447, 84.909, 0, 22.538, 76.197]
  MoveL 7364 to (-14.21, 71.1, -11.5) mm, rotated rx 180 ry 0 rz 90 deg; joints [76.023, -17.873, 86.624, 0, 21.249, 76.023]
  MoveL 7365 to (-15.93, 71.14, -11.5) mm, rotated rx -180 ry 0 rz 90 deg; joints [76.01, -17.903, 86.745, 0, 21.158, 76.01]
  MoveC 7366 to (-18.13, 68.45, -11.5) mm, rotated rx -180 ry 0 rz 90 deg; joints [75.902, -17.928, 86.851, 0, 21.077, 75.902] to (-17.86, 64.99, -11.5) mm, rotated rx 180 ry 0 rz 90 deg; joints [75.789, -17.909, 86.771, 0, 21.138, 75.789]
  MoveL 7367 to (-8.05, 58.64, -11.5) mm, rotated rx 180 ry 0 rz 90 deg; joints [75.661, -17.714, 85.973, 0, 21.741, 75.661]
  MoveL 7368 to (-5.98, 57.25, -11.5) mm, rotated rx -180 ry 0 rz 90 deg; joints [75.632, -17.671, 85.802, 0, 21.869, 75.632]
  MoveC 7369 to (-5.71, 57.13, -11.5) mm, rotated rx 180 ry 0 rz 90 deg; joints [75.631, -17.666, 85.781, 0, 21.885, 75.631] to (-5.42, 57.1, -11.5) mm, rotated rx -180 ry 0 rz 90 deg; joints [75.632, -17.661, 85.76, 0, 21.901, 75.632]
  MoveC 7370 to (11.76, 58.7, -11.5) mm, rotated rx 180 ry 0 rz 90 deg; joints [75.828, -17.361, 84.572, 0, 22.789, 75.828] to (28.9, 60.65, -11.5) mm, rotated rx -180 ry 0 rz 90 deg; joints [76.032, -17.049, 83.375, 0, 23.674, 76.032]
  MoveL 7371 to (30.8, 60.89, -11.5) mm, rotated rx 180 ry 0 rz 90 deg; joints [76.055, -17.014, 83.243, 0, 23.771, 76.055]
  MoveL 7372 to (39.33, 62.1, -11.5) mm, rotated rx -180 ry 0 rz 90 deg; joints [76.162, -16.855, 82.644, 0, 24.21, 76.162]
  MoveL 7373 to (39.67, 62.15, -11.5) mm, rotated rx -180 ry 0 rz 90 deg; joints [76.167, -16.848, 82.62, 0, 24.228, 76.167]
  MoveL 7374 to (39.67, 68.95, -11.5) mm, rotated rx -180 ry 0 rz 90 deg; joints [76.386, -16.88, 82.741, 0, 24.14, 76.386]
  MoveC 7375 to (27.66, 69.68, -11.5) mm, rotated rx -180 ry 0 rz 90 deg; joints [76.315, -17.115, 83.626, 0, 23.489, 76.315] to (15.64, 70.19, -11.5) mm, rotated rx 180 ry 0 rz 90 deg; joints [76.236, -17.342, 84.499, 0, 22.843, 76.236]
  MoveL 7376 to (11.88, 70.32, -11.5) mm, rotated rx 180 ry 0 rz 90 deg; joints [76.21, -17.411, 84.77, 0, 22.642, 76.21]
  MoveL 7377 to (11.62, 62.78, -11.5) mm, rotated rx 180 ry 0 rz 90 deg; joints [75.961, -17.382, 84.655, 0, 22.727, 75.961]
  MoveL 7378 to (11.62, 62.78, -8.5) mm, rotated rx -180 ry 0 rz 90 deg; joints [75.961, -17.536, 84.758, 0, 22.779, 75.961]
  Establecer velocidad (1000.0 mm/s)
  MoveL 7379 to (11.62, 62.78, 10) mm, rotated rx 180 ry 0 rz 90 deg; joints [75.961, -18.483, 85.377, 0, 23.106, 75.961]
  Establecer velocidad (66.7 mm/s)
  MoveL 7380 to (33.78, 17.15, 10) mm, rotated rx -180 ry 0 rz 90 deg; joints [74.672, -17.824, 82.92, 0, 24.904, 74.672]
  MoveL 7381 to (33.78, 17.15, -8.25) mm, rotated rx 180 ry 0 rz 90 deg; joints [74.672, -16.899, 82.307, 0, 24.591, 74.672]
  MoveL 7382 to (33.97, 18.65, -8.66) mm, rotated rx -180 ry 0 rz 90 deg; joints [74.722, -16.882, 82.309, 0, 24.573, 74.722]
  MoveL 7383 to (33.79, 20.16, -9.06) mm, rotated rx -180 ry 0 rz 90 deg; joints [74.769, -16.873, 82.338, 0, 24.535, 74.769]
  MoveL 7384 to (33.29, 21.6, -9.47) mm, rotated rx 180 ry 0 rz 90 deg; joints [74.81, -16.87, 82.389, 0, 24.481, 74.81]
  MoveL 7385 to (32.48, 22.88, -9.88) mm, rotated rx 180 ry 0 rz 90 deg; joints [74.845, -16.872, 82.46, 0, 24.413, 74.845]
  MoveL 7386 to (31.41, 23.96, -10.28) mm, rotated rx -180 ry 0 rz 90 deg; joints [74.87, -16.879, 82.545, 0, 24.334, 74.87]
  MoveL 7387 to (30.12, 24.77, -10.69) mm, rotated rx 180 ry 0 rz 90 deg; joints [74.885, -16.887, 82.64, 0, 24.247, 74.885]
  MoveL 7388 to (28.69, 25.28, -11.09) mm, rotated rx 180 ry 0 rz 90 deg; joints [74.888, -16.897, 82.74, 0, 24.157, 74.888]
  MoveL 7389 to (27.18, 25.42, -11.5) mm, rotated rx 180 ry 0 rz 90 deg; joints [74.88, -16.907, 82.839, 0, 24.068, 74.88]
  MoveC 7390 to (20.94, 25.44, -11.5) mm, rotated rx -180 ry 0 rz 90 deg; joints [74.826, -17.027, 83.29, 0, 23.737, 74.826] to (14.69, 25.42, -11.5) mm, rotated rx -180 ry 0 rz 90 deg; joints [74.771, -17.145, 83.738, 0, 23.406, 74.771]
  MoveC 7391 to (12.29, 24.3, -11.5) mm, rotated rx 180 ry 0 rz 90 deg; joints [74.713, -17.184, 83.888, 0, 23.296, 74.713] to (11.45, 21.8, -11.5) mm, rotated rx 180 ry 0 rz 90 deg; joints [74.625, -17.187, 83.899, 0, 23.288, 74.625]
  MoveL 7392 to (11.6, 21.32, -11.5) mm, rotated rx 180 ry 0 rz 90 deg; joints [74.611, -17.182, 83.879, 0, 23.302, 74.611]
  MoveL 7393 to (15.05, 11.98, -11.5) mm, rotated rx 180 ry 0 rz 90 deg; joints [74.34, -17.068, 83.446, 0, 23.622, 74.34]
  MoveC 7394 to (15.29, 11.41, -11.5) mm, rotated rx -180 ry 0 rz 90 deg; joints [74.324, -17.06, 83.417, 0, 23.643, 74.324] to (15.59, 10.86, -11.5) mm, rotated rx -180 ry 0 rz 90 deg; joints [74.309, -17.052, 83.385, 0, 23.667, 74.309]
  MoveC 7395 to (16.27, 10.21, -11.5) mm, rotated rx 180 ry 0 rz 90 deg; joints [74.294, -17.035, 83.323, 0, 23.713, 74.294] to (17.01, 9.62, -11.5) mm, rotated rx 180 ry 0 rz 90 deg; joints [74.282, -17.018, 83.258, 0, 23.76, 74.282]
  MoveL 7396 to (28.26, 1.34, -11.5) mm, rotated rx 180 ry 0 rz 90 deg; joints [74.119, -16.755, 82.276, 0, 24.479, 74.119]
  MoveC 7397 to (29.02, 0.94, -11.5) mm, rotated rx 180 ry 0 rz 90 deg; joints [74.113, -16.738, 82.213, 0, 24.525, 74.113] to (29.86, 0.79, -11.5) mm, rotated rx -180 ry 0 rz 90 deg; joints [74.116, -16.721, 82.149, 0, 24.572, 74.116]
  MoveC 7398 to (31.63, 1.19, -11.5) mm, rotated rx 180 ry 0 rz 90 deg; joints [74.145, -16.688, 82.028, 0, 24.66, 74.145] to (33, 2.37, -11.5) mm, rotated rx 180 ry 0 rz 90 deg; joints [74.195, -16.667, 81.952, 0, 24.715, 74.195]
  MoveL 7399 to (33.64, 3.28, -11.5) mm, rotated rx 180 ry 0 rz 90 deg; joints [74.229, -16.66, 81.925, 0, 24.735, 74.229]
  MoveL 7400 to (39.67, 12.15, -11.5) mm, rotated rx -180 ry 0 rz 90 deg; joints [74.565, -16.589, 81.665, 0, 24.924, 74.565]
  MoveL 7401 to (39.67, 25.28, -11.5) mm, rotated rx 180 ry 0 rz 90 deg; joints [74.983, -16.66, 81.926, 0, 24.734, 74.983]
  MoveC 7402 to (33.43, 25.37, -11.5) mm, rotated rx 180 ry 0 rz 90 deg; joints [74.932, -16.784, 82.384, 0, 24.4, 74.932] to (27.18, 25.42, -11.5) mm, rotated rx 180 ry 0 rz 90 deg; joints [74.88, -16.907, 82.839, 0, 24.068, 74.88]
  MoveL 7403 to (27.14, 17.87, -11.5) mm, rotated rx -180 ry 0 rz 90 deg; joints [74.637, -16.868, 82.693, 0, 24.175, 74.637]
  MoveL 7404 to (27.14, 17.87, -8.5) mm, rotated rx 180 ry 0 rz 90 deg; joints [74.637, -17.02, 82.795, 0, 24.225, 74.637]
  Establecer velocidad (1000.0 mm/s)
  MoveL 7405 to (27.14, 17.87, 10) mm, rotated rx 180 ry 0 rz 90 deg; joints [74.637, -17.96, 83.416, 0, 24.544, 74.637]
  Establecer velocidad (66.7 mm/s)
  MoveL 7406 to (14.32, -62.23, 10) mm, rotated rx 180 ry 0 rz 90 deg; joints [71.972, -17.738, 82.607, 0, 25.131, 71.972]
  MoveL 7407 to (14.32, -62.23, -8.25) mm, rotated rx -180 ry 0 rz 90 deg; joints [71.972, -16.813, 81.994, 0, 24.819, 71.972]
  MoveL 7408 to (14.19, -63.74, -8.66) mm, rotated rx 180 ry 0 rz 90 deg; joints [71.923, -16.785, 81.954, 0, 24.832, 71.923]
  MoveL 7409 to (14.43, -65.24, -9.06) mm, rotated rx -180 ry 0 rz 90 deg; joints [71.879, -16.75, 81.887, 0, 24.863, 71.879]
  MoveL 7410 to (15, -66.65, -9.47) mm, rotated rx -180 ry 0 rz 90 deg; joints [71.84, -16.709, 81.799, 0, 24.91, 71.84]
  MoveL 7411 to (15.87, -67.9, -9.88) mm, rotated rx 180 ry 0 rz 90 deg; joints [71.81, -16.663, 81.693, 0, 24.971, 71.81]
  MoveL 7412 to (16.99, -68.93, -10.28) mm, rotated rx 180 ry 0 rz 90 deg; joints [71.789, -16.614, 81.574, 0, 25.04, 71.789]
  MoveL 7413 to (18.31, -69.68, -10.69) mm, rotated rx -180 ry 0 rz 90 deg; joints [71.78, -16.562, 81.446, 0, 25.116, 71.78]
  MoveL 7414 to (19.77, -70.12, -11.09) mm, rotated rx -180 ry 0 rz 90 deg; joints [71.781, -16.509, 81.316, 0, 25.193, 71.781]
  MoveL 7415 to (21.28, -70.2, -11.5) mm, rotated rx 180 ry 0 rz 90 deg; joints [71.794, -16.458, 81.191, 0, 25.267, 71.794]
  MoveC 7416 to (27.46, -69.93, -11.5) mm, rotated rx 180 ry 0 rz 90 deg; joints [71.865, -16.334, 80.747, 0, 25.587, 71.865] to (33.64, -69.65, -11.5) mm, rotated rx 180 ry 0 rz 90 deg; joints [71.937, -16.209, 80.302, 0, 25.907, 71.937]
  MoveL 7417 to (39.67, -69.28, -11.5) mm, rotated rx 180 ry 0 rz 90 deg; joints [72.009, -16.086, 79.867, 0, 26.219, 72.009]
  MoveL 7418 to (39.67, -59.65, -11.5) mm, rotated rx 180 ry 0 rz 90 deg; joints [72.308, -16.151, 80.095, 0, 26.055, 72.308]
  MoveC 7419 to (31.4, -49.45, -11.5) mm, rotated rx -180 ry 0 rz 90 deg; joints [72.544, -16.388, 80.94, 0, 25.448, 72.544] to (23.04, -39.33, -11.5) mm, rotated rx 180 ry 0 rz 90 deg; joints [72.78, -16.62, 81.778, 0, 24.841, 72.78]
  MoveL 7420 to (22.27, -38.63, -11.5) mm, rotated rx -180 ry 0 rz 90 deg; joints [72.795, -16.639, 81.85, 0, 24.79, 72.795]
  MoveL 7421 to (13.94, -31.75, -11.5) mm, rotated rx -180 ry 0 rz 90 deg; joints [72.931, -16.844, 82.604, 0, 24.24, 72.931]
  MoveC 7422 to (11.22, -31.18, -11.5) mm, rotated rx -180 ry 0 rz 90 deg; joints [72.923, -16.899, 82.811, 0, 24.088, 72.923] to (8.9, -32.69, -11.5) mm, rotated rx 180 ry 0 rz 90 deg; joints [72.852, -16.935, 82.944, 0, 23.991, 72.852]
  MoveL 7423 to (8.61, -33.64, -11.5) mm, rotated rx -180 ry 0 rz 90 deg; joints [72.819, -16.935, 82.944, 0, 23.99, 72.819]
  MoveL 7424 to (7.11, -39.11, -11.5) mm, rotated rx -180 ry 0 rz 90 deg; joints [72.63, -16.931, 82.93, 0, 24.001, 72.63]
  MoveL 7425 to (-0.47, -67.07, -11.5) mm, rotated rx 180 ry 0 rz 90 deg; joints [71.667, -16.904, 82.829, 0, 24.075, 71.667]
  MoveC 7426 to (-0.56, -67.68, -11.5) mm, rotated rx 180 ry 0 rz 90 deg; joints [71.646, -16.902, 82.82, 0, 24.082, 71.646] to (-0.48, -68.3, -11.5) mm, rotated rx -180 ry 0 rz 90 deg; joints [71.628, -16.896, 82.8, 0, 24.096, 71.628]
  MoveC 7427 to (0.75, -70.15, -11.5) mm, rotated rx -180 ry 0 rz 90 deg; joints [71.582, -16.861, 82.668, 0, 24.193, 71.582] to (2.87, -70.83, -11.5) mm, rotated rx 180 ry 0 rz 90 deg; joints [71.583, -16.816, 82.501, 0, 24.315, 71.583]
  MoveC 7428 to (12.08, -70.54, -11.5) mm, rotated rx -180 ry 0 rz 90 deg; joints [71.688, -16.639, 81.848, 0, 24.791, 71.688] to (21.28, -70.2, -11.5) mm, rotated rx 180 ry 0 rz 90 deg; joints [71.794, -16.458, 81.191, 0, 25.267, 71.794]
  MoveL 7429 to (20.98, -62.65, -11.5) mm, rotated rx 180 ry 0 rz 90 deg; joints [72.027, -16.513, 81.392, 0, 25.122, 72.027]
  MoveL 7430 to (20.98, -62.65, -8.5) mm, rotated rx -180 ry 0 rz 90 deg; joints [72.027, -16.665, 81.494, 0, 25.171, 72.027]
  Establecer velocidad (1000.0 mm/s)
  MoveL 7431 to (20.98, -62.65, 10) mm, rotated rx -180 ry 0 rz 90 deg; joints [72.027, -17.601, 82.116, 0, 25.485, 72.027]
  Establecer velocidad (66.7 mm/s)
  MoveL 7432 to (-37.95, -52.13, 10) mm, rotated rx 180 ry 0 rz 90 deg; joints [71.748, -18.777, 86.521, 0, 22.256, 71.748]
  MoveL 7433 to (-37.95, -52.13, -8.25) mm, rotated rx 180 ry 0 rz 90 deg; joints [71.748, -17.838, 85.911, 0, 21.928, 71.748]
  MoveL 7434 to (-36.54, -52.68, -8.66) mm, rotated rx 180 ry 0 rz 90 deg; joints [71.745, -17.79, 85.787, 0, 22.003, 71.745]
  MoveL 7435 to (-35.03, -52.88, -9.06) mm, rotated rx 180 ry 0 rz 90 deg; joints [71.755, -17.742, 85.665, 0, 22.077, 71.755]
  MoveL 7436 to (-33.52, -52.75, -9.47) mm, rotated rx 180 ry 0 rz 90 deg; joints [71.775, -17.696, 85.549, 0, 22.146, 71.775]
  MoveL 7437 to (-32.08, -52.28, -9.88) mm, rotated rx 180 ry 0 rz 90 deg; joints [71.806, -17.652, 85.446, 0, 22.206, 71.806]
  MoveL 7438 to (-30.77, -51.5, -10.28) mm, rotated rx 180 ry 0 rz 90 deg; joints [71.845, -17.613, 85.359, 0, 22.254, 71.845]
  MoveL 7439 to (-29.67, -50.45, -10.69) mm, rotated rx -180 ry 0 rz 90 deg; joints [71.89, -17.579, 85.293, 0, 22.286, 71.89]
  MoveL 7440 to (-28.83, -49.18, -11.09) mm, rotated rx 180 ry 0 rz 90 deg; joints [71.94, -17.55, 85.249, 0, 22.301, 71.94]
  MoveL 7441 to (-28.32, -47.76, -11.5) mm, rotated rx -180 ry 0 rz 90 deg; joints [71.991, -17.529, 85.232, 0, 22.297, 71.991]
  MoveL 7442 to (-22.83, -26.54, -11.5) mm, rotated rx 180 ry 0 rz 90 deg; joints [72.734, -17.551, 85.32, 0, 22.231, 72.734]
  MoveL 7443 to (-22.67, -25.83, -11.5) mm, rotated rx 180 ry 0 rz 90 deg; joints [72.758, -17.552, 85.324, 0, 22.228, 72.758]
  MoveC 7444 to (-22.63, -25.47, -11.5) mm, rotated rx 180 ry 0 rz 90 deg; joints [72.771, -17.553, 85.329, 0, 22.224, 72.771] to (-22.66, -25.11, -11.5) mm, rotated rx -180 ry 0 rz 90 deg; joints [72.782, -17.556, 85.339, 0, 22.217, 72.782]
  MoveC 7445 to (-23.67, -23.13, -11.5) mm, rotated rx 180 ry 0 rz 90 deg; joints [72.836, -17.584, 85.452, 0, 22.132, 72.836] to (-25.59, -22.02, -11.5) mm, rotated rx -180 ry 0 rz 90 deg; joints [72.853, -17.623, 85.609, 0, 22.014, 72.853]
  MoveC 7446 to (-26, -22.03, -11.5) mm, rotated rx 180 ry 0 rz 90 deg; joints [72.849, -17.631, 85.638, 0, 21.993, 72.849] to (-26.42, -22.08, -11.5) mm, rotated rx -180 ry 0 rz 90 deg; joints [72.842, -17.637, 85.666, 0, 21.972, 72.842]
  MoveC 7447 to (-48.26, -26.53, -11.5) mm, rotated rx -180 ry 0 rz 90 deg; joints [72.474, -17.982, 87.074, 0, 20.908, 72.474] to (-70.09, -31.04, -11.5) mm, rotated rx 180 ry 0 rz 90 deg; joints [72.095, -18.306, 88.455, 0, 19.851, 72.095]
  MoveC 7448 to (-71.26, -31.59, -11.5) mm, rotated rx -180 ry 0 rz 90 deg; joints [72.064, -18.321, 88.521, 0, 19.8, 72.064] to (-72.05, -32.63, -11.5) mm, rotated rx -180 ry 0 rz 90 deg; joints [72.022, -18.328, 88.552, 0, 19.777, 72.022]
  MoveC 7449 to (-72.27, -33.33, -11.5) mm, rotated rx 180 ry 0 rz 90 deg; joints [71.996, -18.328, 88.551, 0, 19.777, 71.996] to (-72.34, -34.06, -11.5) mm, rotated rx 180 ry 0 rz 90 deg; joints [71.971, -18.326, 88.54, 0, 19.785, 71.971]
  MoveL 7450 to (-72.34, -69, -11.5) mm, rotated rx 180 ry 0 rz 90 deg; joints [70.82, -18.143, 87.751, 0, 20.392, 70.82]
  MoveC 7451 to (-71.51, -71.04, -11.5) mm, rotated rx 180 ry 0 rz 90 deg; joints [70.763, -18.118, 87.647, 0, 20.471, 70.763] to (-69.49, -71.92, -11.5) mm, rotated rx 180 ry 0 rz 90 deg; joints [70.757, -18.081, 87.491, 0, 20.59, 70.757]
  MoveC 7452 to (-68.92, -71.92, -11.5) mm, rotated rx 180 ry 0 rz 90 deg; joints [70.763, -18.072, 87.452, 0, 20.62, 70.763] to (-68.35, -71.93, -11.5) mm, rotated rx -180 ry 0 rz 90 deg; joints [70.77, -18.063, 87.414, 0, 20.649, 70.77]
  MoveC 7453 to (-52.5, -71.72, -11.5) mm, rotated rx 180 ry 0 rz 90 deg; joints [70.955, -17.805, 86.344, 0, 21.461, 70.955] to (-36.66, -71.44, -11.5) mm, rotated rx -180 ry 0 rz 90 deg; joints [71.139, -17.537, 85.263, 0, 22.273, 71.139]
  MoveC 7454 to (-35.08, -70.94, -11.5) mm, rotated rx 180 ry 0 rz 90 deg; joints [71.173, -17.512, 85.166, 0, 22.346, 71.173] to (-34.02, -69.67, -11.5) mm, rotated rx -180 ry 0 rz 90 deg; joints [71.225, -17.501, 85.122, 0, 22.379, 71.225]
  MoveC 7455 to (-33.91, -69.4, -11.5) mm, rotated rx -180 ry 0 rz 90 deg; joints [71.235, -17.501, 85.122, 0, 22.379, 71.235] to (-33.83, -69.12, -11.5) mm, rotated rx 180 ry 0 rz 90 deg; joints [71.245, -17.501, 85.122, 0, 22.379, 71.245]
  MoveL 7456 to (-28.32, -47.76, -11.5) mm, rotated rx -180 ry 0 rz 90 deg; joints [71.991, -17.529, 85.232, 0, 22.297, 71.991]
  MoveL 7457 to (-35.63, -45.87, -11.5) mm, rotated rx -180 ry 0 rz 90 deg; joints [71.975, -17.666, 85.781, 0, 21.885, 71.975]
  MoveL 7458 to (-35.63, -45.87, -8.5) mm, rotated rx 180 ry 0 rz 90 deg; joints [71.975, -17.821, 85.883, 0, 21.938, 71.975]
  Establecer velocidad (1000.0 mm/s)
  MoveL 7459 to (-35.63, -45.87, 10) mm, rotated rx 180 ry 0 rz 90 deg; joints [71.975, -18.772, 86.502, 0, 22.27, 71.975]
  Establecer velocidad (66.7 mm/s)
  MoveL 7460 to (-38.1, -52.09, 10) mm, rotated rx 180 ry 0 rz 90 deg; joints [71.748, -18.78, 86.532, 0, 22.248, 71.748]
  MoveL 7461 to (-38.1, -52.09, -8.5) mm, rotated rx 180 ry 0 rz 90 deg; joints [71.748, -17.828, 85.913, 0, 21.915, 71.748]
  MoveL 7462 to (-36.69, -52.65, -8.91) mm, rotated rx 180 ry 0 rz 90 deg; joints [71.745, -17.78, 85.789, 0, 21.991, 71.745]
  MoveL 7463 to (-35.18, -52.85, -9.31) mm, rotated rx -180 ry 0 rz 90 deg; joints [71.754, -17.732, 85.667, 0, 22.065, 71.754]
  MoveL 7464 to (-33.67, -52.71, -9.72) mm, rotated rx 180 ry 0 rz 90 deg; joints [71.775, -17.686, 85.552, 0, 22.134, 71.775]
  MoveL 7465 to (-32.22, -52.24, -10.12) mm, rotated rx -180 ry 0 rz 90 deg; joints [71.806, -17.642, 85.449, 0, 22.194, 71.806]
  MoveL 7466 to (-30.92, -51.46, -10.53) mm, rotated rx -180 ry 0 rz 90 deg; joints [71.844, -17.603, 85.362, 0, 22.241, 71.844]
  MoveL 7467 to (-29.82, -50.41, -10.94) mm, rotated rx 180 ry 0 rz 90 deg; joints [71.89, -17.569, 85.296, 0, 22.273, 71.89]
  MoveL 7468 to (-28.97, -49.15, -11.34) mm, rotated rx -180 ry 0 rz 90 deg; joints [71.94, -17.54, 85.252, 0, 22.289, 71.94]
  MoveL 7469 to (-28.46, -47.72, -11.75) mm, rotated rx 180 ry 0 rz 90 deg; joints [71.991, -17.519, 85.235, 0, 22.284, 71.991]
  MoveL 7470 to (-23.37, -27.96, -11.75) mm, rotated rx -180 ry 0 rz 90 deg; joints [72.683, -17.54, 85.318, 0, 22.222, 72.683]
  MoveL 7471 to (-22.89, -26.06, -11.75) mm, rotated rx 180 ry 0 rz 90 deg; joints [72.749, -17.542, 85.326, 0, 22.216, 72.749]
  MoveL 7472 to (-22.81, -25.59, -11.75) mm, rotated rx 180 ry 0 rz 90 deg; joints [72.765, -17.543, 85.331, 0, 22.212, 72.765]
  MoveC 7473 to (-23.57, -23.7, -11.75) mm, rotated rx 180 ry 0 rz 90 deg; joints [72.818, -17.566, 85.424, 0, 22.142, 72.818] to (-25.15, -22.42, -11.75) mm, rotated rx -180 ry 0 rz 90 deg; joints [72.844, -17.601, 85.561, 0, 22.039, 72.844]
  MoveC 7474 to (-25.78, -22.24, -11.75) mm, rotated rx 180 ry 0 rz 90 deg; joints [72.844, -17.613, 85.609, 0, 22.004, 72.844] to (-26.44, -22.27, -11.75) mm, rotated rx -180 ry 0 rz 90 deg; joints [72.836, -17.624, 85.654, 0, 21.97, 72.836]
  MoveC 7475 to (-48.19, -26.68, -11.75) mm, rotated rx -180 ry 0 rz 90 deg; joints [72.47, -17.967, 87.058, 0, 20.909, 72.47] to (-69.94, -31.16, -11.75) mm, rotated rx -180 ry 0 rz 90 deg; joints [72.093, -18.29, 88.433, 0, 19.857, 72.093]
  MoveC 7476 to (-71.09, -31.7, -11.75) mm, rotated rx 180 ry 0 rz 90 deg; joints [72.063, -18.305, 88.499, 0, 19.806, 72.063] to (-71.88, -32.72, -11.75) mm, rotated rx 180 ry 0 rz 90 deg; joints [72.02, -18.312, 88.53, 0, 19.782, 72.02]
  MoveC 7477 to (-72.1, -33.41, -11.75) mm, rotated rx 180 ry 0 rz 90 deg; joints [71.995, -18.312, 88.53, 0, 19.782, 71.995] to (-72.18, -34.13, -11.75) mm, rotated rx 180 ry 0 rz 90 deg; joints [71.97, -18.31, 88.519, 0, 19.791, 71.97]
  MoveL 7478 to (-72.18, -67.76, -11.75) mm, rotated rx -180 ry 0 rz 90 deg; joints [70.862, -18.134, 87.761, 0, 20.373, 70.862]
  MoveL 7479 to (-72.18, -68.88, -11.75) mm, rotated rx -180 ry 0 rz 90 deg; joints [70.826, -18.128, 87.734, 0, 20.394, 70.826]
  MoveC 7480 to (-71.54, -70.69, -11.75) mm, rotated rx 180 ry 0 rz 90 deg; joints [70.774, -18.108, 87.649, 0, 20.459, 70.774] to (-69.92, -71.71, -11.75) mm, rotated rx 180 ry 0 rz 90 deg; joints [70.759, -18.076, 87.516, 0, 20.56, 70.759]
  MoveC 7481 to (-69.51, -71.78, -11.75) mm, rotated rx 180 ry 0 rz 90 deg; joints [70.761, -18.069, 87.487, 0, 20.583, 70.761] to (-69.09, -71.8, -11.75) mm, rotated rx 180 ry 0 rz 90 deg; joints [70.766, -18.063, 87.458, 0, 20.605, 70.766]
  MoveC 7482 to (-53.04, -71.57, -11.75) mm, rotated rx -180 ry 0 rz 90 deg; joints [70.954, -17.802, 86.376, 0, 21.426, 70.954] to (-36.99, -71.3, -11.75) mm, rotated rx -180 ry 0 rz 90 deg; joints [71.14, -17.53, 85.281, 0, 22.25, 71.14]
  MoveC 7483 to (-36.68, -71.29, -11.75) mm, rotated rx -180 ry 0 rz 90 deg; joints [71.144, -17.525, 85.26, 0, 22.265, 71.144] to (-36.37, -71.25, -11.75) mm, rotated rx 180 ry 0 rz 90 deg; joints [71.149, -17.52, 85.24, 0, 22.28, 71.149]
  MoveC 7484 to (-34.84, -70.51, -11.75) mm, rotated rx 180 ry 0 rz 90 deg; joints [71.189, -17.498, 85.151, 0, 22.347, 71.189] to (-33.97, -69.06, -11.75) mm, rotated rx 180 ry 0 rz 90 deg; joints [71.245, -17.491, 85.125, 0, 22.366, 71.245]
  MoveL 7485 to (-28.46, -47.72, -11.75) mm, rotated rx 180 ry 0 rz 90 deg; joints [71.991, -17.519, 85.235, 0, 22.284, 71.991]
  MoveL 7486 to (-35.77, -45.83, -11.75) mm, rotated rx 180 ry 0 rz 90 deg; joints [71.975, -17.656, 85.783, 0, 21.873, 71.975]
  MoveL 7487 to (-35.77, -45.83, -8.75) mm, rotated rx -180 ry 0 rz 90 deg; joints [71.975, -17.811, 85.886, 0, 21.925, 71.975]
  Establecer velocidad (1000.0 mm/s)
  MoveL 7488 to (-35.77, -45.83, 10) mm, rotated rx -180 ry 0 rz 90 deg; joints [71.975, -18.775, 86.513, 0, 22.262, 71.975]
  Establecer velocidad (66.7 mm/s)
  MoveL 7489 to (12.97, -62.08, 10) mm, rotated rx 180 ry 0 rz 90 deg; joints [71.963, -17.766, 82.708, 0, 25.058, 71.963]
  MoveL 7490 to (12.97, -62.08, -8.5) mm, rotated rx -180 ry 0 rz 90 deg; joints [71.963, -16.828, 82.086, 0, 24.742, 71.963]
  MoveL 7491 to (12.85, -63.6, -8.91) mm, rotated rx -180 ry 0 rz 90 deg; joints [71.914, -16.8, 82.045, 0, 24.755, 71.914]
  MoveL 7492 to (13.09, -65.1, -9.31) mm, rotated rx 180 ry 0 rz 90 deg; joints [71.869, -16.765, 81.979, 0, 24.787, 71.869]
  MoveL 7493 to (13.67, -66.5, -9.72) mm, rotated rx 180 ry 0 rz 90 deg; joints [71.831, -16.724, 81.89, 0, 24.834, 71.831]
  MoveL 7494 to (14.53, -67.75, -10.12) mm, rotated rx -180 ry 0 rz 90 deg; joints [71.801, -16.678, 81.784, 0, 24.894, 71.801]
  MoveL 7495 to (15.66, -68.77, -10.53) mm, rotated rx 180 ry 0 rz 90 deg; joints [71.781, -16.629, 81.665, 0, 24.964, 71.781]
  MoveL 7496 to (16.98, -69.52, -10.94) mm, rotated rx -180 ry 0 rz 90 deg; joints [71.771, -16.577, 81.538, 0, 25.039, 71.771]
  MoveL 7497 to (18.44, -69.96, -11.34) mm, rotated rx 180 ry 0 rz 90 deg; joints [71.772, -16.524, 81.408, 0, 25.116, 71.772]
  MoveL 7498 to (19.95, -70.03, -11.75) mm, rotated rx 180 ry 0 rz 90 deg; joints [71.785, -16.473, 81.282, 0, 25.191, 71.785]
  MoveC 7499 to (28.39, -69.64, -11.75) mm, rotated rx 180 ry 0 rz 90 deg; joints [71.884, -16.305, 80.678, 0, 25.627, 71.884] to (36.82, -69.19, -11.75) mm, rotated rx -180 ry 0 rz 90 deg; joints [71.983, -16.134, 80.071, 0, 26.063, 71.983]
  MoveL 7500 to (36.82, -56.53, -11.75) mm, rotated rx -180 ry 0 rz 90 deg; joints [72.377, -16.218, 80.37, 0, 25.848, 72.377]
  MoveL 7501 to (35.19, -54.49, -11.75) mm, rotated rx -180 ry 0 rz 90 deg; joints [72.424, -16.265, 80.537, 0, 25.728, 72.424]
  MoveL 7502 to (26.06, -43.32, -11.75) mm, rotated rx 180 ry 0 rz 90 deg; joints [72.684, -16.522, 81.46, 0, 25.062, 72.684]
  MoveL 7503 to (23.22, -39.86, -11.75) mm, rotated rx -180 ry 0 rz 90 deg; joints [72.765, -16.6, 81.745, 0, 24.855, 72.765]
  MoveL 7504 to (22.72, -39.33, -11.75) mm, rotated rx 180 ry 0 rz 90 deg; joints [72.777, -16.613, 81.793, 0, 24.82, 72.777]
  MoveL 7505 to (22.27, -38.92, -11.75) mm, rotated rx 180 ry 0 rz 90 deg; joints [72.786, -16.625, 81.835, 0, 24.79, 72.786]
  MoveL 7506 to (14.69, -32.64, -11.75) mm, rotated rx -180 ry 0 rz 90 deg; joints [72.91, -16.811, 82.522, 0, 24.289, 72.91]
  MoveL 7507 to (14.22, -32.24, -11.75) mm, rotated rx -180 ry 0 rz 90 deg; joints [72.918, -16.823, 82.565, 0, 24.258, 72.918]
  MoveL 7508 to (13.74, -31.88, -11.75) mm, rotated rx 180 ry 0 rz 90 deg; joints [72.925, -16.834, 82.607, 0, 24.227, 72.925]
  MoveC 7509 to (11.17, -31.57, -11.75) mm, rotated rx 180 ry 0 rz 90 deg; joints [72.91, -16.885, 82.798, 0, 24.087, 72.91] to (9.03, -33.03, -11.75) mm, rotated rx 180 ry 0 rz 90 deg; joints [72.842, -16.918, 82.919, 0, 23.999, 72.842]
  MoveL 7510 to (7.55, -38.38, -11.75) mm, rotated rx -180 ry 0 rz 90 deg; joints [72.658, -16.914, 82.906, 0, 24.008, 72.658]
  MoveL 7511 to (-0.22, -67, -11.75) mm, rotated rx -180 ry 0 rz 90 deg; joints [71.671, -16.887, 82.804, 0, 24.083, 71.671]
  MoveC 7512 to (-0.28, -67.36, -11.75) mm, rotated rx 180 ry 0 rz 90 deg; joints [71.659, -16.886, 82.8, 0, 24.086, 71.659] to (-0.28, -67.73, -11.75) mm, rotated rx -180 ry 0 rz 90 deg; joints [71.648, -16.883, 82.79, 0, 24.093, 71.648]
  MoveC 7513 to (0.84, -69.82, -11.75) mm, rotated rx -180 ry 0 rz 90 deg; joints [71.593, -16.849, 82.662, 0, 24.187, 71.593] to (3.07, -70.62, -11.75) mm, rotated rx 180 ry 0 rz 90 deg; joints [71.592, -16.801, 82.483, 0, 24.318, 71.592]
  MoveC 7514 to (11.51, -70.36, -11.75) mm, rotated rx 180 ry 0 rz 90 deg; joints [71.688, -16.638, 81.884, 0, 24.754, 71.688] to (19.95, -70.03, -11.75) mm, rotated rx 180 ry 0 rz 90 deg; joints [71.785, -16.473, 81.282, 0, 25.191, 71.785]
  MoveL 7515 to (19.63, -62.49, -11.75) mm, rotated rx -180 ry 0 rz 90 deg; joints [72.018, -16.529, 81.484, 0, 25.044, 72.018]
  MoveL 7516 to (19.63, -62.49, -8.75) mm, rotated rx -180 ry 0 rz 90 deg; joints [72.018, -16.681, 81.587, 0, 25.094, 72.018]
  Establecer velocidad (1000.0 mm/s)
  MoveL 7517 to (19.63, -62.49, 10) mm, rotated rx -180 ry 0 rz 90 deg; joints [72.018, -17.629, 82.218, 0, 25.412, 72.018]
  Establecer velocidad (66.7 mm/s)
  MoveL 7518 to (32.5, 16.91, 10) mm, rotated rx 180 ry 0 rz 90 deg; joints [74.654, -17.848, 83.008, 0, 24.84, 74.654]
  MoveL 7519 to (32.5, 16.91, -8.5) mm, rotated rx 180 ry 0 rz 90 deg; joints [74.654, -16.91, 82.387, 0, 24.523, 74.654]
  MoveL 7520 to (32.69, 18.42, -8.91) mm, rotated rx 180 ry 0 rz 90 deg; joints [74.704, -16.894, 82.389, 0, 24.505, 74.704]
  MoveL 7521 to (32.52, 19.93, -9.31) mm, rotated rx 180 ry 0 rz 90 deg; joints [74.75, -16.885, 82.418, 0, 24.467, 74.75]
  MoveL 7522 to (32.02, 21.36, -9.72) mm, rotated rx 180 ry 0 rz 90 deg; joints [74.792, -16.882, 82.469, 0, 24.413, 74.792]
  MoveL 7523 to (31.21, 22.65, -10.12) mm, rotated rx -180 ry 0 rz 90 deg; joints [74.826, -16.884, 82.539, 0, 24.344, 74.826]
  MoveL 7524 to (30.14, 23.73, -10.53) mm, rotated rx -180 ry 0 rz 90 deg; joints [74.851, -16.89, 82.624, 0, 24.265, 74.851]
  MoveL 7525 to (28.85, 24.54, -10.94) mm, rotated rx -180 ry 0 rz 90 deg; joints [74.866, -16.898, 82.72, 0, 24.179, 74.866]
  MoveL 7526 to (27.42, 25.05, -11.34) mm, rotated rx 180 ry 0 rz 90 deg; joints [74.87, -16.908, 82.819, 0, 24.089, 74.87]
  MoveL 7527 to (25.91, 25.19, -11.75) mm, rotated rx 180 ry 0 rz 90 deg; joints [74.862, -16.917, 82.918, 0, 24, 74.862]
  MoveC 7528 to (20.46, 25.21, -11.75) mm, rotated rx -180 ry 0 rz 90 deg; joints [74.815, -17.022, 83.312, 0, 23.71, 74.815] to (15, 25.2, -11.75) mm, rotated rx 180 ry 0 rz 90 deg; joints [74.766, -17.125, 83.703, 0, 23.422, 74.766]
  MoveC 7529 to (12.98, 24.48, -11.75) mm, rotated rx 180 ry 0 rz 90 deg; joints [74.725, -17.159, 83.834, 0, 23.326, 74.725] to (11.85, 22.67, -11.75) mm, rotated rx 180 ry 0 rz 90 deg; joints [74.657, -17.171, 83.879, 0, 23.292, 74.657]
  MoveL 7530 to (11.79, 22.42, -11.75) mm, rotated rx 180 ry 0 rz 90 deg; joints [74.648, -17.171, 83.879, 0, 23.292, 74.648]
  MoveC 7531 to (11.73, 21.86, -11.75) mm, rotated rx -180 ry 0 rz 90 deg; joints [74.63, -17.169, 83.872, 0, 23.297, 74.63] to (11.85, 21.32, -11.75) mm, rotated rx -180 ry 0 rz 90 deg; joints [74.613, -17.164, 83.853, 0, 23.311, 74.613]
  MoveL 7532 to (15.41, 11.7, -11.75) mm, rotated rx -180 ry 0 rz 90 deg; joints [74.334, -17.047, 83.406, 0, 23.641, 74.334]
  MoveC 7533 to (15.79, 11, -11.75) mm, rotated rx -180 ry 0 rz 90 deg; joints [74.315, -17.036, 83.365, 0, 23.671, 74.315] to (16.36, 10.43, -11.75) mm, rotated rx 180 ry 0 rz 90 deg; joints [74.302, -17.022, 83.313, 0, 23.709, 74.302]
  MoveL 7534 to (17.53, 9.54, -11.75) mm, rotated rx 180 ry 0 rz 90 deg; joints [74.284, -16.995, 83.21, 0, 23.785, 74.284]
  MoveL 7535 to (28.22, 1.67, -11.75) mm, rotated rx 180 ry 0 rz 90 deg; joints [74.129, -16.745, 82.277, 0, 24.468, 74.129]
  MoveC 7536 to (29.72, 1.11, -11.75) mm, rotated rx 180 ry 0 rz 90 deg; joints [74.125, -16.713, 82.157, 0, 24.555, 74.125] to (31.28, 1.42, -11.75) mm, rotated rx 180 ry 0 rz 90 deg; joints [74.149, -16.684, 82.05, 0, 24.633, 74.149]
  MoveC 7537 to (32.15, 1.84, -11.75) mm, rotated rx 180 ry 0 rz 90 deg; joints [74.17, -16.669, 81.996, 0, 24.673, 74.17] to (32.83, 2.52, -11.75) mm, rotated rx -180 ry 0 rz 90 deg; joints [74.198, -16.659, 81.96, 0, 24.699, 74.198]
  MoveL 7538 to (33.39, 3.32, -11.75) mm, rotated rx -180 ry 0 rz 90 deg; joints [74.228, -16.652, 81.935, 0, 24.717, 74.228]
  MoveL 7539 to (36.82, 8.36, -11.75) mm, rotated rx 180 ry 0 rz 90 deg; joints [74.419, -16.612, 81.788, 0, 24.824, 74.419]
  MoveL 7540 to (36.82, 25.06, -11.75) mm, rotated rx 180 ry 0 rz 90 deg; joints [74.952, -16.703, 82.123, 0, 24.581, 74.952]
  MoveC 7541 to (31.36, 25.15, -11.75) mm, rotated rx 180 ry 0 rz 90 deg; joints [74.907, -16.811, 82.521, 0, 24.29, 74.907] to (25.91, 25.19, -11.75) mm, rotated rx 180 ry 0 rz 90 deg; joints [74.862, -16.917, 82.918, 0, 24, 74.862]
  MoveL 7542 to (25.86, 17.65, -11.75) mm, rotated rx -180 ry 0 rz 90 deg; joints [74.619, -16.878, 82.772, 0, 24.106, 74.619]
  MoveL 7543 to (25.86, 17.65, -8.75) mm, rotated rx -180 ry 0 rz 90 deg; joints [74.619, -17.031, 82.874, 0, 24.157, 74.619]
  Establecer velocidad (1000.0 mm/s)
  MoveL 7544 to (25.86, 17.65, 10) mm, rotated rx 180 ry 0 rz 90 deg; joints [74.619, -17.984, 83.504, 0, 24.48, 74.619]
  Establecer velocidad (66.7 mm/s)
  MoveL 7545 to (-3.84, 59.72, 10) mm, rotated rx -180 ry 0 rz 90 deg; joints [75.732, -18.751, 86.417, 0, 22.333, 75.732]
  MoveL 7546 to (-3.84, 59.72, -8.5) mm, rotated rx 180 ry 0 rz 90 deg; joints [75.732, -17.8, 85.798, 0, 22.001, 75.732]
  MoveL 7547 to (-2.68, 58.74, -8.91) mm, rotated rx 180 ry 0 rz 90 deg; joints [75.709, -17.754, 85.685, 0, 22.069, 75.709]
  MoveL 7548 to (-1.31, 58.09, -9.31) mm, rotated rx -180 ry 0 rz 90 deg; joints [75.7, -17.706, 85.563, 0, 22.143, 75.7]
  MoveL 7549 to (0.18, 57.78, -9.72) mm, rotated rx 180 ry 0 rz 90 deg; joints [75.702, -17.657, 85.438, 0, 22.219, 75.702]
  MoveL 7550 to (1.7, 57.84, -10.12) mm, rotated rx 180 ry 0 rz 90 deg; joints [75.717, -17.609, 85.318, 0, 22.291, 75.717]
  MoveL 7551 to (3.16, 58.25, -10.53) mm, rotated rx -180 ry 0 rz 90 deg; joints [75.742, -17.564, 85.208, 0, 22.356, 75.742]
  MoveL 7552 to (4.48, 59, -10.94) mm, rotated rx -180 ry 0 rz 90 deg; joints [75.778, -17.523, 85.114, 0, 22.409, 75.778]
  MoveL 7553 to (5.59, 60.04, -11.34) mm, rotated rx 180 ry 0 rz 90 deg; joints [75.821, -17.487, 85.04, 0, 22.447, 75.821]
  MoveL 7554 to (6.4, 61.33, -11.75) mm, rotated rx -180 ry 0 rz 90 deg; joints [75.87, -17.457, 84.992, 0, 22.465, 75.87]
  MoveL 7555 to (10.76, 70.16, -11.75) mm, rotated rx 180 ry 0 rz 90 deg; joints [76.196, -17.418, 84.838, 0, 22.58, 76.196]
  MoveL 7556 to (2.37, 70.43, -11.75) mm, rotated rx 180 ry 0 rz 90 deg; joints [76.137, -17.57, 85.439, 0, 22.131, 76.137]
  MoveL 7557 to (-14.21, 70.91, -11.75) mm, rotated rx -180 ry 0 rz 90 deg; joints [76.017, -17.86, 86.613, 0, 21.247, 76.017]
  MoveL 7558 to (-15.31, 70.94, -11.75) mm, rotated rx 180 ry 0 rz 90 deg; joints [76.008, -17.878, 86.69, 0, 21.189, 76.008]
  MoveC 7559 to (-17.48, 68.28, -11.75) mm, rotated rx -180 ry 0 rz 90 deg; joints [75.902, -17.904, 86.794, 0, 21.109, 75.902] to (-17.22, 64.86, -11.75) mm, rotated rx 180 ry 0 rz 90 deg; joints [75.79, -17.885, 86.716, 0, 21.169, 75.79]
  MoveL 7560 to (-7.11, 58.28, -11.75) mm, rotated rx 180 ry 0 rz 90 deg; joints [75.657, -17.683, 85.892, 0, 21.791, 75.657]
  MoveL 7561 to (-5.64, 57.31, -11.75) mm, rotated rx 180 ry 0 rz 90 deg; joints [75.637, -17.653, 85.771, 0, 21.882, 75.637]
  MoveC 7562 to (-5.49, 57.25, -11.75) mm, rotated rx 180 ry 0 rz 90 deg; joints [75.636, -17.65, 85.759, 0, 21.891, 75.636] to (-5.33, 57.23, -11.75) mm, rotated rx -180 ry 0 rz 90 deg; joints [75.637, -17.647, 85.748, 0, 21.899, 75.637]
  MoveC 7563 to (11.8, 58.86, -11.75) mm, rotated rx 180 ry 0 rz 90 deg; joints [75.834, -17.348, 84.563, 0, 22.785, 75.834] to (28.9, 60.84, -11.75) mm, rotated rx -180 ry 0 rz 90 deg; joints [76.038, -17.037, 83.37, 0, 23.667, 76.038]
  MoveL 7564 to (29.85, 60.97, -11.75) mm, rotated rx 180 ry 0 rz 90 deg; joints [76.05, -17.02, 83.304, 0, 23.716, 76.05]
  MoveL 7565 to (36.82, 61.95, -11.75) mm, rotated rx -180 ry 0 rz 90 deg; joints [76.138, -16.89, 82.816, 0, 24.074, 76.138]
  MoveL 7566 to (36.82, 68.9, -11.75) mm, rotated rx 180 ry 0 rz 90 deg; joints [76.362, -16.923, 82.94, 0, 23.983, 76.362]
  MoveC 7567 to (24.2, 69.61, -11.75) mm, rotated rx 180 ry 0 rz 90 deg; joints [76.286, -17.168, 83.866, 0, 23.302, 76.286] to (11.58, 70.13, -11.75) mm, rotated rx -180 ry 0 rz 90 deg; joints [76.201, -17.403, 84.779, 0, 22.624, 76.201]
  MoveL 7568 to (10.76, 70.16, -11.75) mm, rotated rx 180 ry 0 rz 90 deg; joints [76.196, -17.418, 84.838, 0, 22.58, 76.196]
  MoveL 7569 to (10.52, 62.61, -11.75) mm, rotated rx -180 ry 0 rz 90 deg; joints [75.946, -17.389, 84.722, 0, 22.666, 75.946]
  MoveL 7570 to (10.52, 62.61, -8.75) mm, rotated rx 180 ry 0 rz 90 deg; joints [75.946, -17.543, 84.825, 0, 22.718, 75.946]
  Establecer velocidad (1000.0 mm/s)
  MoveL 7571 to (10.52, 62.61, 10) mm, rotated rx 180 ry 0 rz 90 deg; joints [75.946, -18.503, 85.453, 0, 23.05, 75.946]
  Establecer velocidad (66.7 mm/s)
  MoveL 7572 to (-63.94, 35.92, 10) mm, rotated rx 180 ry 0 rz 90 deg; joints [74.401, -19.643, 90.118, 0, 19.525, 74.401]
  MoveL 7573 to (-63.94, 35.92, -8.5) mm, rotated rx -180 ry 0 rz 90 deg; joints [74.401, -18.676, 89.499, 0, 19.177, 74.401]
  MoveL 7574 to (-65.45, 36.11, -8.91) mm, rotated rx 180 ry 0 rz 90 deg; joints [74.393, -18.678, 89.59, 0, 19.089, 74.393]
  MoveL 7575 to (-66.95, 35.92, -9.31) mm, rotated rx 180 ry 0 rz 90 deg; joints [74.373, -18.679, 89.674, 0, 19.005, 74.373]
  MoveL 7576 to (-68.38, 35.41, -9.72) mm, rotated rx 180 ry 0 rz 90 deg; joints [74.342, -18.676, 89.746, 0, 18.93, 74.342]
  MoveL 7577 to (-69.67, 34.59, -10.12) mm, rotated rx -180 ry 0 rz 90 deg; joints [74.302, -18.671, 89.803, 0, 18.868, 74.302]
  MoveL 7578 to (-70.74, 33.52, -10.53) mm, rotated rx 180 ry 0 rz 90 deg; joints [74.255, -18.661, 89.84, 0, 18.82, 74.255]
  MoveL 7579 to (-71.54, 32.23, -10.94) mm, rotated rx -180 ry 0 rz 90 deg; joints [74.203, -18.646, 89.856, 0, 18.79, 74.203]
  MoveL 7580 to (-72.04, 30.79, -11.34) mm, rotated rx -180 ry 0 rz 90 deg; joints [74.15, -18.626, 89.848, 0, 18.777, 74.15]
  MoveL 7581 to (-72.18, 29.28, -11.75) mm, rotated rx -180 ry 0 rz 90 deg; joints [74.097, -18.6, 89.815, 0, 18.785, 74.097]
  MoveL 7582 to (-72.18, 3.32, -11.75) mm, rotated rx 180 ry 0 rz 90 deg; joints [73.221, -18.488, 89.306, 0, 19.182, 73.221]
  MoveC 7583 to (-71.08, 0.93, -11.75) mm, rotated rx -180 ry 0 rz 90 deg; joints [73.152, -18.46, 89.184, 0, 19.277, 73.152] to (-68.52, 0.34, -11.75) mm, rotated rx -180 ry 0 rz 90 deg; joints [73.158, -18.419, 89, 0, 19.419, 73.158]
  MoveC 7584 to (-46.33, 5.58, -11.75) mm, rotated rx 180 ry 0 rz 90 deg; joints [73.554, -18.097, 87.604, 0, 20.493, 73.554] to (-24.17, 10.92, -11.75) mm, rotated rx -180 ry 0 rz 90 deg; joints [73.943, -17.755, 86.184, 0, 21.571, 73.943]
  MoveL 7585 to (-23.22, 11.3, -11.75) mm, rotated rx 180 ry 0 rz 90 deg; joints [73.965, -17.741, 86.126, 0, 21.615, 73.965]
  MoveL 7586 to (-23.11, 11.37, -11.75) mm, rotated rx 180 ry 0 rz 90 deg; joints [73.968, -17.739, 86.12, 0, 21.619, 73.968]
  MoveC 7587 to (-22, 12.85, -11.75) mm, rotated rx -180 ry 0 rz 90 deg; joints [74.027, -17.728, 86.073, 0, 21.655, 74.027] to (-21.84, 14.69, -11.75) mm, rotated rx -180 ry 0 rz 90 deg; joints [74.089, -17.734, 86.098, 0, 21.636, 74.089]
  MoveL 7588 to (-22.15, 15.64, -11.75) mm, rotated rx 180 ry 0 rz 90 deg; joints [74.117, -17.744, 86.138, 0, 21.606, 74.117]
  MoveL 7589 to (-27.19, 29.85, -11.75) mm, rotated rx -180 ry 0 rz 90 deg; joints [74.54, -17.897, 86.764, 0, 21.132, 74.54]
  MoveL 7590 to (-27.51, 30.71, -11.75) mm, rotated rx -180 ry 0 rz 90 deg; joints [74.565, -17.906, 86.803, 0, 21.103, 74.565]
  MoveC 7591 to (-27.98, 31.52, -11.75) mm, rotated rx 180 ry 0 rz 90 deg; joints [74.588, -17.918, 86.852, 0, 21.066, 74.588] to (-28.68, 32.16, -11.75) mm, rotated rx -180 ry 0 rz 90 deg; joints [74.602, -17.932, 86.912, 0, 21.02, 74.602]
  MoveC 7592 to (-48.32, 44.98, -11.75) mm, rotated rx -180 ry 0 rz 90 deg; joints [74.852, -18.305, 88.5, 0, 19.806, 74.852] to (-68.01, 57.73, -11.75) mm, rotated rx -180 ry 0 rz 90 deg; joints [75.105, -18.654, 90.061, 0, 18.593, 75.105]
  MoveC 7593 to (-70.33, 57.5, -11.75) mm, rotated rx 180 ry 0 rz 90 deg; joints [75.076, -18.687, 90.212, 0, 18.475, 75.076] to (-72.02, 55.9, -11.75) mm, rotated rx 180 ry 0 rz 90 deg; joints [75.006, -18.705, 90.296, 0, 18.409, 75.006]
  MoveC 7594 to (-72.14, 55.58, -11.75) mm, rotated rx -180 ry 0 rz 90 deg; joints [74.994, -18.705, 90.298, 0, 18.407, 74.994] to (-72.18, 55.25, -11.75) mm, rotated rx 180 ry 0 rz 90 deg; joints [74.982, -18.705, 90.295, 0, 18.41, 74.982]
  MoveL 7595 to (-72.18, 29.28, -11.75) mm, rotated rx -180 ry 0 rz 90 deg; joints [74.097, -18.6, 89.815, 0, 18.785, 74.097]
  MoveL 7596 to (-64.63, 29.28, -11.75) mm, rotated rx 180 ry 0 rz 90 deg; joints [74.17, -18.488, 89.309, 0, 19.18, 74.17]
  MoveL 7597 to (-64.63, 29.28, -8.75) mm, rotated rx 180 ry 0 rz 90 deg; joints [74.17, -18.645, 89.411, 0, 19.234, 74.17]
  Establecer velocidad (1000.0 mm/s)
  MoveL 7598 to (-64.63, 29.28, 10) mm, rotated rx 180 ry 0 rz 90 deg; joints [74.17, -19.625, 90.039, 0, 19.586, 74.17]
  Establecer velocidad (66.7 mm/s)
  MoveL 7599 to (-63.78, 35.92, 10) mm, rotated rx 180 ry 0 rz 90 deg; joints [74.403, -19.641, 90.107, 0, 19.534, 74.403]
  MoveL 7600 to (-63.78, 35.92, -8.75) mm, rotated rx -180 ry 0 rz 90 deg; joints [74.403, -18.661, 89.479, 0, 19.181, 74.403]
  MoveL 7601 to (-65.28, 36.11, -9.16) mm, rotated rx -180 ry 0 rz 90 deg; joints [74.395, -18.663, 89.57, 0, 19.093, 74.395]
  MoveL 7602 to (-66.79, 35.92, -9.56) mm, rotated rx -180 ry 0 rz 90 deg; joints [74.374, -18.663, 89.654, 0, 19.009, 74.374]
  MoveL 7603 to (-68.22, 35.41, -9.97) mm, rotated rx -180 ry 0 rz 90 deg; joints [74.343, -18.661, 89.727, 0, 18.934, 74.343]
  MoveL 7604 to (-69.5, 34.59, -10.38) mm, rotated rx -180 ry 0 rz 90 deg; joints [74.303, -18.655, 89.783, 0, 18.872, 74.303]
  MoveL 7605 to (-70.57, 33.52, -10.78) mm, rotated rx 180 ry 0 rz 90 deg; joints [74.256, -18.645, 89.821, 0, 18.824, 74.256]
  MoveL 7606 to (-71.38, 32.23, -11.19) mm, rotated rx 180 ry 0 rz 90 deg; joints [74.205, -18.63, 89.836, 0, 18.794, 74.205]
  MoveL 7607 to (-71.88, 30.79, -11.59) mm, rotated rx 180 ry 0 rz 90 deg; joints [74.152, -18.61, 89.829, 0, 18.782, 74.152]
  MoveL 7608 to (-72.02, 29.28, -12) mm, rotated rx 180 ry 0 rz 90 deg; joints [74.099, -18.585, 89.796, 0, 18.789, 74.099]
  MoveL 7609 to (-72.02, 3.32, -12) mm, rotated rx 180 ry 0 rz 90 deg; joints [73.222, -18.472, 89.286, 0, 19.186, 73.222]
  MoveC 7610 to (-71.91, 2.53, -12) mm, rotated rx -180 ry 0 rz 90 deg; joints [73.197, -18.467, 89.263, 0, 19.204, 73.197] to (-71.55, 1.82, -12) mm, rotated rx 180 ry 0 rz 90 deg; joints [73.177, -18.458, 89.225, 0, 19.234, 73.177]
  MoveC 7611 to (-70.32, 0.72, -12) mm, rotated rx 180 ry 0 rz 90 deg; joints [73.152, -18.435, 89.12, 0, 19.315, 73.152] to (-68.7, 0.44, -12) mm, rotated rx 180 ry 0 rz 90 deg; joints [73.159, -18.409, 89.006, 0, 19.403, 73.159]
  MoveC 7612 to (-46.66, 5.66, -12) mm, rotated rx 180 ry 0 rz 90 deg; joints [73.553, -18.09, 87.62, 0, 20.47, 73.553] to (-24.64, 10.97, -12) mm, rotated rx -180 ry 0 rz 90 deg; joints [73.941, -17.751, 86.21, 0, 21.541, 73.941]
  MoveL 7613 to (-24.17, 11.1, -12) mm, rotated rx -180 ry 0 rz 90 deg; joints [73.949, -17.743, 86.179, 0, 21.564, 73.949]
  MoveL 7614 to (-23.48, 11.37, -12) mm, rotated rx -180 ry 0 rz 90 deg; joints [73.965, -17.733, 86.137, 0, 21.595, 73.965]
  MoveC 7615 to (-22.77, 12.01, -12) mm, rotated rx -180 ry 0 rz 90 deg; joints [73.992, -17.724, 86.101, 0, 21.623, 73.992] to (-22.27, 12.81, -12) mm, rotated rx -180 ry 0 rz 90 deg; joints [74.024, -17.719, 86.082, 0, 21.637, 74.024]
  MoveL 7616 to (-22.06, 13.53, -12) mm, rotated rx 180 ry 0 rz 90 deg; joints [74.049, -17.719, 86.081, 0, 21.638, 74.049]
  MoveC 7617 to (-21.96, 14.28, -12) mm, rotated rx 180 ry 0 rz 90 deg; joints [74.075, -17.721, 86.09, 0, 21.631, 74.075] to (-22.1, 15.04, -12) mm, rotated rx 180 ry 0 rz 90 deg; joints [74.098, -17.727, 86.114, 0, 21.613, 74.098]
  MoveL 7618 to (-27.5, 30.28, -12) mm, rotated rx 180 ry 0 rz 90 deg; joints [74.551, -17.891, 86.786, 0, 21.105, 74.551]
  MoveC 7619 to (-27.7, 30.77, -12) mm, rotated rx 180 ry 0 rz 90 deg; joints [74.565, -17.897, 86.809, 0, 21.087, 74.565] to (-27.96, 31.23, -12) mm, rotated rx 180 ry 0 rz 90 deg; joints [74.578, -17.903, 86.836, 0, 21.067, 74.578]
  MoveC 7620 to (-28.39, 31.71, -12) mm, rotated rx -180 ry 0 rz 90 deg; joints [74.59, -17.912, 86.875, 0, 21.038, 74.59] to (-28.9, 32.11, -12) mm, rotated rx -180 ry 0 rz 90 deg; joints [74.599, -17.923, 86.918, 0, 21.005, 74.599]
  MoveC 7621 to (-48.37, 44.83, -12) mm, rotated rx 180 ry 0 rz 90 deg; joints [74.846, -18.292, 88.491, 0, 19.801, 74.846] to (-67.88, 57.48, -12) mm, rotated rx -180 ry 0 rz 90 deg; joints [75.098, -18.638, 90.039, 0, 18.599, 75.098]
  MoveC 7622 to (-70.05, 57.31, -12) mm, rotated rx -180 ry 0 rz 90 deg; joints [75.072, -18.669, 90.181, 0, 18.488, 75.072] to (-71.72, 55.91, -12) mm, rotated rx 180 ry 0 rz 90 deg; joints [75.009, -18.688, 90.268, 0, 18.42, 75.009]
  MoveC 7623 to (-71.94, 55.46, -12) mm, rotated rx -180 ry 0 rz 90 deg; joints [74.991, -18.689, 90.275, 0, 18.414, 74.991] to (-72.02, 54.96, -12) mm, rotated rx 180 ry 0 rz 90 deg; joints [74.974, -18.688, 90.271, 0, 18.417, 74.974]
  MoveL 7624 to (-72.02, 29.28, -12) mm, rotated rx 180 ry 0 rz 90 deg; joints [74.099, -18.585, 89.796, 0, 18.789, 74.099]
  MoveL 7625 to (-64.47, 29.28, -12) mm, rotated rx -180 ry 0 rz 90 deg; joints [74.172, -18.473, 89.289, 0, 19.184, 74.172]
  MoveL 7626 to (-64.47, 29.28, -9) mm, rotated rx -180 ry 0 rz 90 deg; joints [74.172, -18.63, 89.391, 0, 19.238, 74.172]
  Establecer velocidad (1000.0 mm/s)
  MoveL 7627 to (-64.47, 29.28, 10) mm, rotated rx 180 ry 0 rz 90 deg; joints [74.172, -19.623, 90.028, 0, 19.595, 74.172]
  Establecer velocidad (66.7 mm/s)
  MoveL 7628 to (-8.11, 65.56, 10) mm, rotated rx -180 ry 0 rz 90 deg; joints [75.89, -18.853, 86.821, 0, 22.032, 75.89]
  MoveL 7629 to (-8.11, 65.56, -8.75) mm, rotated rx 180 ry 0 rz 90 deg; joints [75.89, -17.887, 86.194, 0, 21.693, 75.89]
  MoveL 7630 to (-8.33, 64.06, -9.16) mm, rotated rx 180 ry 0 rz 90 deg; joints [75.838, -17.863, 86.169, 0, 21.694, 75.838]
  MoveL 7631 to (-8.16, 62.55, -9.56) mm, rotated rx -180 ry 0 rz 90 deg; joints [75.789, -17.833, 86.116, 0, 21.717, 75.789]
  MoveL 7632 to (-7.64, 61.13, -9.97) mm, rotated rx 180 ry 0 rz 90 deg; joints [75.747, -17.797, 86.04, 0, 21.756, 75.747]
  MoveL 7633 to (-6.79, 59.87, -10.38) mm, rotated rx 180 ry 0 rz 90 deg; joints [75.712, -17.755, 85.945, 0, 21.811, 75.712]
  MoveL 7634 to (-5.67, 58.84, -10.78) mm, rotated rx -180 ry 0 rz 90 deg; joints [75.688, -17.71, 85.833, 0, 21.877, 75.688]
  MoveL 7635 to (-4.34, 58.11, -11.19) mm, rotated rx -180 ry 0 rz 90 deg; joints [75.675, -17.663, 85.713, 0, 21.95, 75.675]
  MoveL 7636 to (-2.87, 57.71, -11.59) mm, rotated rx -180 ry 0 rz 90 deg; joints [75.674, -17.614, 85.588, 0, 22.026, 75.674]
  MoveL 7637 to (-1.35, 57.71, -12) mm, rotated rx 180 ry 0 rz 90 deg; joints [75.687, -17.567, 85.467, 0, 22.099, 75.687]
  MoveL 7638 to (7.67, 58.57, -12) mm, rotated rx 180 ry 0 rz 90 deg; joints [75.79, -17.409, 84.844, 0, 22.565, 75.79]
  MoveC 7639 to (18.63, 59.77, -12) mm, rotated rx -180 ry 0 rz 90 deg; joints [75.92, -17.213, 84.082, 0, 23.131, 75.92] to (29.59, 61.12, -12) mm, rotated rx -180 ry 0 rz 90 deg; joints [76.053, -17.013, 83.318, 0, 23.696, 76.053]
  MoveL 7640 to (33.96, 61.75, -12) mm, rotated rx 180 ry 0 rz 90 deg; joints [76.108, -16.932, 83.012, 0, 23.92, 76.108]
  MoveL 7641 to (33.96, 68.85, -12) mm, rotated rx 180 ry 0 rz 90 deg; joints [76.338, -16.966, 83.138, 0, 23.827, 76.338]
  MoveC 7642 to (18.17, 69.66, -12) mm, rotated rx -180 ry 0 rz 90 deg; joints [76.239, -17.267, 84.291, 0, 22.976, 76.239] to (2.37, 70.24, -12) mm, rotated rx 180 ry 0 rz 90 deg; joints [76.13, -17.556, 85.427, 0, 22.13, 76.13]
  MoveL 7643 to (-14.69, 70.74, -12) mm, rotated rx -180 ry 0 rz 90 deg; joints [76.007, -17.854, 86.634, 0, 21.22, 76.007]
  MoveC 7644 to (-16.83, 68.11, -12) mm, rotated rx -180 ry 0 rz 90 deg; joints [75.901, -17.879, 86.738, 0, 21.141, 75.901] to (-16.58, 64.73, -12) mm, rotated rx -180 ry 0 rz 90 deg; joints [75.791, -17.861, 86.661, 0, 21.2, 75.791]
  MoveL 7645 to (-8.05, 59.19, -12) mm, rotated rx 180 ry 0 rz 90 deg; joints [75.679, -17.691, 85.966, 0, 21.725, 75.679]
  MoveL 7646 to (-5.78, 57.67, -12) mm, rotated rx 180 ry 0 rz 90 deg; joints [75.648, -17.644, 85.778, 0, 21.866, 75.648]
  MoveC 7647 to (-5.5, 57.5, -12) mm, rotated rx -180 ry 0 rz 90 deg; joints [75.645, -17.639, 85.756, 0, 21.882, 75.645] to (-5.21, 57.37, -12) mm, rotated rx 180 ry 0 rz 90 deg; joints [75.643, -17.633, 85.733, 0, 21.9, 75.643]
  MoveC 7648 to (1.23, 57.94, -12) mm, rotated rx 180 ry 0 rz 90 deg; joints [75.716, -17.522, 85.289, 0, 22.233, 75.716] to (7.67, 58.57, -12) mm, rotated rx 180 ry 0 rz 90 deg; joints [75.79, -17.409, 84.844, 0, 22.565, 75.79]
  MoveL 7649 to (6.9, 66.09, -12) mm, rotated rx -180 ry 0 rz 90 deg; joints [76.031, -17.457, 85.033, 0, 22.424, 76.031]
  MoveL 7650 to (6.9, 66.09, -9) mm, rotated rx 180 ry 0 rz 90 deg; joints [76.031, -17.611, 85.135, 0, 22.476, 76.031]
  Establecer velocidad (1000.0 mm/s)
  MoveL 7651 to (6.9, 66.09, 10) mm, rotated rx 180 ry 0 rz 90 deg; joints [76.031, -18.585, 85.771, 0, 22.814, 76.031]
  Establecer velocidad (66.7 mm/s)
  MoveL 7652 to (25.72, 8.07, 10) mm, rotated rx 180 ry 0 rz 90 deg; joints [74.311, -17.934, 83.322, 0, 24.613, 74.311]
  MoveL 7653 to (25.72, 8.07, -8.75) mm, rotated rx 180 ry 0 rz 90 deg; joints [74.311, -16.982, 82.692, 0, 24.29, 74.311]
  MoveL 7654 to (27.23, 7.89, -9.16) mm, rotated rx 180 ry 0 rz 90 deg; joints [74.319, -16.931, 82.566, 0, 24.365, 74.319]
  MoveL 7655 to (28.74, 8.07, -9.56) mm, rotated rx -180 ry 0 rz 90 deg; joints [74.338, -16.882, 82.446, 0, 24.436, 74.338]
  MoveL 7656 to (30.17, 8.59, -9.97) mm, rotated rx -180 ry 0 rz 90 deg; joints [74.367, -16.836, 82.339, 0, 24.497, 74.367]
  MoveL 7657 to (31.45, 9.4, -10.38) mm, rotated rx 180 ry 0 rz 90 deg; joints [74.405, -16.794, 82.248, 0, 24.546, 74.405]
  MoveL 7658 to (32.52, 10.48, -10.78) mm, rotated rx 180 ry 0 rz 90 deg; joints [74.449, -16.759, 82.178, 0, 24.58, 74.449]
  MoveL 7659 to (33.32, 11.77, -11.19) mm, rotated rx -180 ry 0 rz 90 deg; joints [74.497, -16.729, 82.132, 0, 24.597, 74.497]
  MoveL 7660 to (33.82, 13.21, -11.59) mm, rotated rx 180 ry 0 rz 90 deg; joints [74.547, -16.707, 82.111, 0, 24.596, 74.547]
  MoveL 7661 to (33.96, 14.71, -12) mm, rotated rx 180 ry 0 rz 90 deg; joints [74.596, -16.691, 82.117, 0, 24.574, 74.596]
  MoveL 7662 to (33.96, 24.85, -12) mm, rotated rx 180 ry 0 rz 90 deg; joints [74.921, -16.746, 82.318, 0, 24.428, 74.921]
  MoveL 7663 to (31.75, 24.9, -12) mm, rotated rx 180 ry 0 rz 90 deg; joints [74.903, -16.79, 82.48, 0, 24.309, 74.903]
  MoveL 7664 to (16.58, 24.99, -12) mm, rotated rx 180 ry 0 rz 90 deg; joints [74.774, -17.081, 83.577, 0, 23.504, 74.774]
  MoveL 7665 to (15.28, 24.98, -12) mm, rotated rx 180 ry 0 rz 90 deg; joints [74.762, -17.106, 83.67, 0, 23.436, 74.762]
  MoveC 7666 to (12.86, 23.87, -12) mm, rotated rx -180 ry 0 rz 90 deg; joints [74.705, -17.146, 83.822, 0, 23.324, 74.705] to (12.1, 21.32, -12) mm, rotated rx -180 ry 0 rz 90 deg; joints [74.615, -17.147, 83.826, 0, 23.32, 74.615]
  MoveL 7667 to (15.61, 11.85, -12) mm, rotated rx 180 ry 0 rz 90 deg; joints [74.341, -17.031, 83.386, 0, 23.645, 74.341]
  MoveC 7668 to (16, 11.13, -12) mm, rotated rx -180 ry 0 rz 90 deg; joints [74.321, -17.02, 83.344, 0, 23.676, 74.321] to (16.58, 10.55, -12) mm, rotated rx -180 ry 0 rz 90 deg; joints [74.308, -17.006, 83.29, 0, 23.716, 74.308]
  MoveL 7669 to (17.37, 9.95, -12) mm, rotated rx 180 ry 0 rz 90 deg; joints [74.296, -16.988, 83.222, 0, 23.766, 74.296]
  MoveL 7670 to (28.25, 1.97, -12) mm, rotated rx -180 ry 0 rz 90 deg; joints [74.139, -16.734, 82.273, 0, 24.461, 74.139]
  MoveC 7671 to (28.98, 1.59, -12) mm, rotated rx 180 ry 0 rz 90 deg; joints [74.133, -16.717, 82.212, 0, 24.505, 74.133] to (29.79, 1.45, -12) mm, rotated rx 180 ry 0 rz 90 deg; joints [74.136, -16.7, 82.15, 0, 24.55, 74.136]
  MoveC 7672 to (31.59, 1.88, -12) mm, rotated rx 180 ry 0 rz 90 deg; joints [74.166, -16.667, 82.028, 0, 24.639, 74.166] to (32.97, 3.11, -12) mm, rotated rx -180 ry 0 rz 90 deg; joints [74.218, -16.647, 81.953, 0, 24.694, 74.218]
  MoveL 7673 to (33.96, 4.58, -12) mm, rotated rx 180 ry 0 rz 90 deg; joints [74.273, -16.635, 81.911, 0, 24.724, 74.273]
  MoveL 7674 to (33.96, 14.71, -12) mm, rotated rx 180 ry 0 rz 90 deg; joints [74.596, -16.691, 82.117, 0, 24.574, 74.596]
  MoveL 7675 to (26.41, 14.71, -12) mm, rotated rx -180 ry 0 rz 90 deg; joints [74.53, -16.839, 82.665, 0, 24.174, 74.53]
  MoveL 7676 to (26.41, 14.71, -9) mm, rotated rx 180 ry 0 rz 90 deg; joints [74.53, -16.992, 82.768, 0, 24.224, 74.53]
  Establecer velocidad (1000.0 mm/s)
  MoveL 7677 to (26.41, 14.71, 10) mm, rotated rx 180 ry 0 rz 90 deg; joints [74.53, -17.957, 83.406, 0, 24.552, 74.53]
  Establecer velocidad (66.7 mm/s)
  MoveL 7678 to (11.66, -61.91, 10) mm, rotated rx 180 ry 0 rz 90 deg; joints [71.955, -17.793, 82.806, 0, 24.987, 71.955]
  MoveL 7679 to (11.66, -61.91, -8.75) mm, rotated rx -180 ry 0 rz 90 deg; joints [71.955, -16.842, 82.176, 0, 24.666, 71.955]
  MoveL 7680 to (11.54, -63.42, -9.16) mm, rotated rx 180 ry 0 rz 90 deg; joints [71.906, -16.814, 82.135, 0, 24.679, 71.906]
  MoveL 7681 to (11.79, -64.92, -9.56) mm, rotated rx 180 ry 0 rz 90 deg; joints [71.861, -16.779, 82.068, 0, 24.711, 71.861]
  MoveL 7682 to (12.36, -66.33, -9.97) mm, rotated rx 180 ry 0 rz 90 deg; joints [71.823, -16.738, 81.98, 0, 24.758, 71.823]
  MoveL 7683 to (13.23, -67.58, -10.38) mm, rotated rx 180 ry 0 rz 90 deg; joints [71.793, -16.692, 81.874, 0, 24.818, 71.793]
  MoveL 7684 to (14.35, -68.6, -10.78) mm, rotated rx 180 ry 0 rz 90 deg; joints [71.772, -16.643, 81.755, 0, 24.888, 71.772]
  MoveL 7685 to (15.67, -69.35, -11.19) mm, rotated rx -180 ry 0 rz 90 deg; joints [71.763, -16.591, 81.628, 0, 24.964, 71.763]
  MoveL 7686 to (17.13, -69.79, -11.59) mm, rotated rx 180 ry 0 rz 90 deg; joints [71.764, -16.539, 81.498, 0, 25.041, 71.764]
  MoveL 7687 to (18.64, -69.86, -12) mm, rotated rx 180 ry 0 rz 90 deg; joints [71.777, -16.488, 81.373, 0, 25.115, 71.777]
  MoveC 7688 to (26.3, -69.51, -12) mm, rotated rx 180 ry 0 rz 90 deg; joints [71.867, -16.336, 80.825, 0, 25.511, 71.867] to (33.96, -69.11, -12) mm, rotated rx 180 ry 0 rz 90 deg; joints [71.957, -16.181, 80.274, 0, 25.907, 71.957]
  MoveL 7689 to (33.96, -53.35, -12) mm, rotated rx -180 ry 0 rz 90 deg; joints [72.448, -16.285, 80.645, 0, 25.64, 72.448]
  MoveL 7690 to (32.58, -51.65, -12) mm, rotated rx -180 ry 0 rz 90 deg; joints [72.487, -16.325, 80.786, 0, 25.539, 72.487]
  MoveL 7691 to (23.24, -40.22, -12) mm, rotated rx 180 ry 0 rz 90 deg; joints [72.754, -16.585, 81.727, 0, 24.858, 72.754]
  MoveC 7692 to (22.64, -39.56, -12) mm, rotated rx -180 ry 0 rz 90 deg; joints [72.769, -16.601, 81.785, 0, 24.816, 72.769] to (21.99, -38.96, -12) mm, rotated rx -180 ry 0 rz 90 deg; joints [72.781, -16.617, 81.845, 0, 24.772, 72.781]
  MoveL 7693 to (14.1, -32.42, -12) mm, rotated rx 180 ry 0 rz 90 deg; joints [72.912, -16.811, 82.56, 0, 24.251, 72.912]
  MoveC 7694 to (11.7, -31.86, -12) mm, rotated rx -180 ry 0 rz 90 deg; joints [72.906, -16.861, 82.745, 0, 24.116, 72.906] to (9.48, -32.93, -12) mm, rotated rx 180 ry 0 rz 90 deg; joints [72.85, -16.897, 82.881, 0, 24.016, 72.85]
  MoveC 7695 to (9.26, -33.21, -12) mm, rotated rx 180 ry 0 rz 90 deg; joints [72.839, -16.9, 82.89, 0, 24.009, 72.839] to (9.12, -33.55, -12) mm, rotated rx 180 ry 0 rz 90 deg; joints [72.827, -16.9, 82.893, 0, 24.007, 72.827]
  MoveL 7696 to (7.53, -39.33, -12) mm, rotated rx -180 ry 0 rz 90 deg; joints [72.627, -16.896, 82.878, 0, 24.018, 72.627]
  MoveL 7697 to (0.06, -66.81, -12) mm, rotated rx -180 ry 0 rz 90 deg; joints [71.68, -16.87, 82.779, 0, 24.091, 71.68]
  MoveC 7698 to (0.84, -69.38, -12) mm, rotated rx 180 ry 0 rz 90 deg; joints [71.607, -16.839, 82.663, 0, 24.176, 71.607] to (3.32, -70.41, -12) mm, rotated rx 180 ry 0 rz 90 deg; joints [71.601, -16.785, 82.462, 0, 24.323, 71.601]
  MoveC 7699 to (10.98, -70.16, -12) mm, rotated rx 180 ry 0 rz 90 deg; joints [71.689, -16.637, 81.919, 0, 24.719, 71.689] to (18.64, -69.86, -12) mm, rotated rx 180 ry 0 rz 90 deg; joints [71.777, -16.488, 81.373, 0, 25.115, 71.777]
  MoveL 7700 to (18.32, -62.32, -12) mm, rotated rx -180 ry 0 rz 90 deg; joints [72.01, -16.543, 81.575, 0, 24.969, 72.01]
  MoveL 7701 to (18.32, -62.32, -9) mm, rotated rx -180 ry 0 rz 90 deg; joints [72.01, -16.695, 81.677, 0, 25.018, 72.01]
  Establecer velocidad (1000.0 mm/s)
  MoveL 7702 to (18.32, -62.32, 10) mm, rotated rx 180 ry 0 rz 90 deg; joints [72.01, -17.657, 82.316, 0, 25.341, 72.01]
  Establecer velocidad (66.7 mm/s)
  MoveL 7703 to (-38.23, -52.01, 10) mm, rotated rx -180 ry 0 rz 90 deg; joints [71.749, -18.783, 86.544, 0, 22.239, 71.749]
  MoveL 7704 to (-38.23, -52.01, -8.75) mm, rotated rx -180 ry 0 rz 90 deg; joints [71.749, -17.818, 85.916, 0, 21.902, 71.749]
  MoveL 7705 to (-36.82, -52.57, -9.16) mm, rotated rx 180 ry 0 rz 90 deg; joints [71.746, -17.77, 85.792, 0, 21.978, 71.746]
  MoveL 7706 to (-35.32, -52.77, -9.56) mm, rotated rx -180 ry 0 rz 90 deg; joints [71.756, -17.722, 85.67, 0, 22.052, 71.756]
  MoveL 7707 to (-33.8, -52.63, -9.97) mm, rotated rx -180 ry 0 rz 90 deg; joints [71.776, -17.675, 85.554, 0, 22.121, 71.776]
  MoveL 7708 to (-32.36, -52.16, -10.38) mm, rotated rx -180 ry 0 rz 90 deg; joints [71.807, -17.632, 85.451, 0, 22.181, 71.807]
  MoveL 7709 to (-31.05, -51.38, -10.78) mm, rotated rx 180 ry 0 rz 90 deg; joints [71.846, -17.593, 85.365, 0, 22.228, 71.846]
  MoveL 7710 to (-29.95, -50.33, -11.19) mm, rotated rx 180 ry 0 rz 90 deg; joints [71.891, -17.559, 85.298, 0, 22.261, 71.891]
  MoveL 7711 to (-29.11, -49.07, -11.59) mm, rotated rx -180 ry 0 rz 90 deg; joints [71.941, -17.53, 85.254, 0, 22.276, 71.941]
  MoveL 7712 to (-28.6, -47.64, -12) mm, rotated rx 180 ry 0 rz 90 deg; joints [71.992, -17.509, 85.237, 0, 22.271, 71.992]
  MoveL 7713 to (-23.13, -26.42, -12) mm, rotated rx -180 ry 0 rz 90 deg; joints [72.735, -17.531, 85.326, 0, 22.205, 72.735]
  MoveC 7714 to (-23.06, -25.72, -12) mm, rotated rx 180 ry 0 rz 90 deg; joints [72.758, -17.534, 85.336, 0, 22.197, 72.758] to (-23.19, -25.02, -12) mm, rotated rx 180 ry 0 rz 90 deg; joints [72.779, -17.54, 85.361, 0, 22.179, 72.779]
  MoveC 7715 to (-23.95, -23.71, -12) mm, rotated rx 180 ry 0 rz 90 deg; joints [72.814, -17.56, 85.442, 0, 22.118, 72.814] to (-25.11, -22.74, -12) mm, rotated rx -180 ry 0 rz 90 deg; joints [72.834, -17.586, 85.544, 0, 22.042, 72.834]
  MoveC 7716 to (-25.8, -22.48, -12) mm, rotated rx 180 ry 0 rz 90 deg; joints [72.836, -17.599, 85.597, 0, 22.002, 72.836] to (-26.54, -22.47, -12) mm, rotated rx 180 ry 0 rz 90 deg; joints [72.829, -17.612, 85.648, 0, 21.963, 72.829]
  MoveC 7717 to (-48.15, -26.84, -12) mm, rotated rx 180 ry 0 rz 90 deg; joints [72.465, -17.953, 87.043, 0, 20.91, 72.465] to (-69.75, -31.27, -12) mm, rotated rx 180 ry 0 rz 90 deg; joints [72.091, -18.274, 88.41, 0, 19.864, 72.091]
  MoveC 7718 to (-71.17, -32.03, -12) mm, rotated rx -180 ry 0 rz 90 deg; joints [72.051, -18.292, 88.488, 0, 19.803, 72.051] to (-71.93, -33.45, -12) mm, rotated rx 180 ry 0 rz 90 deg; joints [71.995, -18.296, 88.509, 0, 19.787, 71.995]
  MoveC 7719 to (-71.99, -33.84, -12) mm, rotated rx -180 ry 0 rz 90 deg; joints [71.982, -18.295, 88.504, 0, 19.791, 71.982] to (-72.02, -34.24, -12) mm, rotated rx -180 ry 0 rz 90 deg; joints [71.968, -18.294, 88.497, 0, 19.796, 71.968]
  MoveL 7720 to (-72.02, -67.76, -12) mm, rotated rx -180 ry 0 rz 90 deg; joints [70.864, -18.118, 87.741, 0, 20.377, 70.864]
  MoveL 7721 to (-72.01, -68.7, -12) mm, rotated rx 180 ry 0 rz 90 deg; joints [70.833, -18.113, 87.719, 0, 20.394, 70.833]
  MoveC 7722 to (-71.36, -70.58, -12) mm, rotated rx -180 ry 0 rz 90 deg; joints [70.779, -18.092, 87.631, 0, 20.462, 70.779] to (-69.65, -71.61, -12) mm, rotated rx -180 ry 0 rz 90 deg; joints [70.765, -18.06, 87.492, 0, 20.568, 70.765]
  MoveC 7723 to (-69.4, -71.64, -12) mm, rotated rx 180 ry 0 rz 90 deg; joints [70.767, -18.056, 87.474, 0, 20.581, 70.767] to (-69.15, -71.65, -12) mm, rotated rx -180 ry 0 rz 90 deg; joints [70.77, -18.051, 87.457, 0, 20.594, 70.77]
  MoveC 7724 to (-53.04, -71.42, -12) mm, rotated rx 180 ry 0 rz 90 deg; joints [70.959, -17.79, 86.371, 0, 21.419, 70.959] to (-36.94, -71.14, -12) mm, rotated rx 180 ry 0 rz 90 deg; joints [71.146, -17.518, 85.273, 0, 22.245, 71.146]
  MoveC 7725 to (-36.1, -71.01, -12) mm, rotated rx 180 ry 0 rz 90 deg; joints [71.159, -17.504, 85.218, 0, 22.286, 71.159] to (-35.33, -70.66, -12) mm, rotated rx 180 ry 0 rz 90 deg; joints [71.179, -17.493, 85.173, 0, 22.32, 71.179]
  MoveC 7726 to (-34.54, -69.87, -12) mm, rotated rx -180 ry 0 rz 90 deg; joints [71.213, -17.483, 85.136, 0, 22.347, 71.213] to (-34.07, -68.85, -12) mm, rotated rx -180 ry 0 rz 90 deg; joints [71.251, -17.481, 85.128, 0, 22.353, 71.251]
  MoveL 7727 to (-28.6, -47.64, -12) mm, rotated rx 180 ry 0 rz 90 deg; joints [71.992, -17.509, 85.237, 0, 22.271, 71.992]
  MoveL 7728 to (-35.91, -45.76, -12) mm, rotated rx -180 ry 0 rz 90 deg; joints [71.976, -17.646, 85.786, 0, 21.86, 71.976]
  MoveL 7729 to (-35.91, -45.76, -9) mm, rotated rx -180 ry 0 rz 90 deg; joints [71.976, -17.801, 85.888, 0, 21.912, 71.976]
  Establecer velocidad (1000.0 mm/s)
  MoveL 7730 to (-35.91, -45.76, 10) mm, rotated rx -180 ry 0 rz 90 deg; joints [71.976, -18.778, 86.524, 0, 22.254, 71.976]
  Establecer velocidad (66.7 mm/s)
  MoveL 7731 to (-38.38, -51.98, 10) mm, rotated rx -180 ry 0 rz 90 deg; joints [71.748, -18.786, 86.554, 0, 22.231, 71.748]
  MoveL 7732 to (-38.38, -51.98, -9) mm, rotated rx -180 ry 0 rz 90 deg; joints [71.748, -17.808, 85.918, 0, 21.89, 71.748]
  MoveL 7733 to (-36.96, -52.53, -9.41) mm, rotated rx 180 ry 0 rz 90 deg; joints [71.745, -17.76, 85.794, 0, 21.966, 71.745]
  MoveL 7734 to (-35.46, -52.73, -9.81) mm, rotated rx 180 ry 0 rz 90 deg; joints [71.755, -17.712, 85.672, 0, 22.04, 71.755]
  MoveL 7735 to (-33.94, -52.59, -10.22) mm, rotated rx -180 ry 0 rz 90 deg; joints [71.776, -17.665, 85.556, 0, 22.109, 71.776]
  MoveL 7736 to (-32.5, -52.12, -10.62) mm, rotated rx 180 ry 0 rz 90 deg; joints [71.806, -17.622, 85.453, 0, 22.169, 71.806]
  MoveL 7737 to (-31.2, -51.34, -11.03) mm, rotated rx 180 ry 0 rz 90 deg; joints [71.845, -17.583, 85.367, 0, 22.216, 71.845]
  MoveL 7738 to (-30.09, -50.29, -11.44) mm, rotated rx 180 ry 0 rz 90 deg; joints [71.891, -17.549, 85.3, 0, 22.248, 71.891]
  MoveL 7739 to (-29.25, -49.03, -11.84) mm, rotated rx -180 ry 0 rz 90 deg; joints [71.94, -17.52, 85.257, 0, 22.264, 71.94]
  MoveL 7740 to (-28.74, -47.6, -12.25) mm, rotated rx 180 ry 0 rz 90 deg; joints [71.992, -17.499, 85.24, 0, 22.259, 71.992]
  MoveL 7741 to (-23.3, -26.43, -12.25) mm, rotated rx -180 ry 0 rz 90 deg; joints [72.733, -17.521, 85.329, 0, 22.192, 72.733]
  MoveC 7742 to (-23.24, -26.02, -12.25) mm, rotated rx -180 ry 0 rz 90 deg; joints [72.746, -17.522, 85.334, 0, 22.188, 72.746] to (-23.29, -25.61, -12.25) mm, rotated rx -180 ry 0 rz 90 deg; joints [72.759, -17.525, 85.346, 0, 22.179, 72.759]
  MoveC 7743 to (-24.12, -23.95, -12.25) mm, rotated rx 180 ry 0 rz 90 deg; joints [72.805, -17.549, 85.44, 0, 22.109, 72.805] to (-25.61, -22.82, -12.25) mm, rotated rx -180 ry 0 rz 90 deg; joints [72.827, -17.581, 85.568, 0, 22.013, 72.827]
  MoveC 7744 to (-26.16, -22.67, -12.25) mm, rotated rx -180 ry 0 rz 90 deg; joints [72.826, -17.591, 85.609, 0, 21.982, 72.826] to (-26.73, -22.69, -12.25) mm, rotated rx -180 ry 0 rz 90 deg; joints [72.82, -17.601, 85.648, 0, 21.953, 72.82]
  MoveC 7745 to (-48.19, -27.01, -12.25) mm, rotated rx 180 ry 0 rz 90 deg; joints [72.459, -17.94, 87.034, 0, 20.906, 72.459] to (-69.64, -31.4, -12.25) mm, rotated rx 180 ry 0 rz 90 deg; joints [72.088, -18.258, 88.391, 0, 19.867, 72.088]
  MoveC 7746 to (-71.15, -32.29, -12.25) mm, rotated rx 180 ry 0 rz 90 deg; joints [72.042, -18.277, 88.473, 0, 19.804, 72.042] to (-71.81, -33.91, -12.25) mm, rotated rx 180 ry 0 rz 90 deg; joints [71.982, -18.279, 88.482, 0, 19.797, 71.982]
  MoveL 7747 to (-71.85, -34.59, -12.25) mm, rotated rx -180 ry 0 rz 90 deg; joints [71.959, -18.276, 88.47, 0, 19.806, 71.959]
  MoveL 7748 to (-71.85, -67.76, -12.25) mm, rotated rx -180 ry 0 rz 90 deg; joints [70.866, -18.103, 87.721, 0, 20.381, 70.866]
  MoveL 7749 to (-71.85, -68.64, -12.25) mm, rotated rx 180 ry 0 rz 90 deg; joints [70.837, -18.098, 87.7, 0, 20.397, 70.837]
  MoveC 7750 to (-70.98, -70.68, -12.25) mm, rotated rx 180 ry 0 rz 90 deg; joints [70.78, -18.073, 87.595, 0, 20.478, 70.78] to (-68.93, -71.51, -12.25) mm, rotated rx -180 ry 0 rz 90 deg; joints [70.777, -18.036, 87.437, 0, 20.599, 70.777]
  MoveC 7751 to (-52.99, -71.27, -12.25) mm, rotated rx -180 ry 0 rz 90 deg; joints [70.964, -17.777, 86.363, 0, 21.415, 70.964] to (-37.05, -70.98, -12.25) mm, rotated rx -180 ry 0 rz 90 deg; joints [71.15, -17.508, 85.275, 0, 22.232, 71.15]
  MoveC 7752 to (-36.62, -70.94, -12.25) mm, rotated rx -180 ry 0 rz 90 deg; joints [71.156, -17.5, 85.247, 0, 22.254, 71.156] to (-36.2, -70.85, -12.25) mm, rotated rx -180 ry 0 rz 90 deg; joints [71.163, -17.494, 85.22, 0, 22.274, 71.163]
  MoveC 7753 to (-35.14, -70.29, -12.25) mm, rotated rx -180 ry 0 rz 90 deg; joints [71.193, -17.479, 85.16, 0, 22.318, 71.193] to (-34.43, -69.33, -12.25) mm, rotated rx 180 ry 0 rz 90 deg; joints [71.232, -17.472, 85.133, 0, 22.339, 71.232]
  MoveC 7754 to (-34.25, -68.87, -12.25) mm, rotated rx 180 ry 0 rz 90 deg; joints [71.248, -17.471, 85.131, 0, 22.34, 71.248] to (-34.1, -68.4, -12.25) mm, rotated rx 180 ry 0 rz 90 deg; joints [71.265, -17.472, 85.132, 0, 22.339, 71.265]
  MoveL 7755 to (-32.69, -62.96, -12.25) mm, rotated rx 180 ry 0 rz 90 deg; joints [71.455, -17.479, 85.162, 0, 22.317, 71.455]
  MoveL 7756 to (-28.74, -47.6, -12.25) mm, rotated rx 180 ry 0 rz 90 deg; joints [71.992, -17.499, 85.24, 0, 22.259, 71.992]
  MoveL 7757 to (-36.06, -45.72, -12.25) mm, rotated rx -180 ry 0 rz 90 deg; joints [71.976, -17.636, 85.788, 0, 21.847, 71.976]
  MoveL 7758 to (-36.06, -45.72, -9.25) mm, rotated rx 180 ry 0 rz 90 deg; joints [71.976, -17.79, 85.891, 0, 21.9, 71.976]
  Establecer velocidad (1000.0 mm/s)
  MoveL 7759 to (-36.06, -45.72, 10) mm, rotated rx -180 ry 0 rz 90 deg; joints [71.976, -18.781, 86.535, 0, 22.245, 71.976]
  Establecer velocidad (66.7 mm/s)
  MoveL 7760 to (10.34, -61.76, 10) mm, rotated rx -180 ry 0 rz 90 deg; joints [71.946, -17.82, 82.904, 0, 24.916, 71.946]
  MoveL 7761 to (10.34, -61.76, -9) mm, rotated rx 180 ry 0 rz 90 deg; joints [71.946, -16.856, 82.266, 0, 24.59, 71.946]
  MoveL 7762 to (10.22, -63.27, -9.41) mm, rotated rx -180 ry 0 rz 90 deg; joints [71.897, -16.828, 82.225, 0, 24.603, 71.897]
  MoveL 7763 to (10.46, -64.77, -9.81) mm, rotated rx -180 ry 0 rz 90 deg; joints [71.853, -16.793, 82.158, 0, 24.635, 71.853]
  MoveL 7764 to (11.04, -66.17, -10.22) mm, rotated rx -180 ry 0 rz 90 deg; joints [71.814, -16.752, 82.07, 0, 24.682, 71.814]
  MoveL 7765 to (11.91, -67.42, -10.62) mm, rotated rx 180 ry 0 rz 90 deg; joints [71.784, -16.707, 81.964, 0, 24.743, 71.784]
  MoveL 7766 to (13.03, -68.44, -11.03) mm, rotated rx -180 ry 0 rz 90 deg; joints [71.764, -16.657, 81.845, 0, 24.812, 71.764]
  MoveL 7767 to (14.36, -69.19, -11.44) mm, rotated rx -180 ry 0 rz 90 deg; joints [71.754, -16.606, 81.718, 0, 24.888, 71.754]
  MoveL 7768 to (15.81, -69.62, -11.84) mm, rotated rx -180 ry 0 rz 90 deg; joints [71.755, -16.553, 81.589, 0, 24.965, 71.755]
  MoveL 7769 to (17.33, -69.7, -12.25) mm, rotated rx 180 ry 0 rz 90 deg; joints [71.769, -16.502, 81.463, 0, 25.039, 71.769]
  MoveC 7770 to (24.21, -69.38, -12.25) mm, rotated rx 180 ry 0 rz 90 deg; joints [71.85, -16.366, 80.971, 0, 25.395, 71.85] to (31.1, -69.01, -12.25) mm, rotated rx -180 ry 0 rz 90 deg; joints [71.931, -16.228, 80.477, 0, 25.751, 71.931]
  MoveL 7771 to (31.1, -50.22, -12.25) mm, rotated rx -180 ry 0 rz 90 deg; joints [72.517, -16.351, 80.918, 0, 25.433, 72.517]
  MoveL 7772 to (24.55, -42.17, -12.25) mm, rotated rx -180 ry 0 rz 90 deg; joints [72.705, -16.534, 81.579, 0, 24.955, 72.705]
  MoveL 7773 to (23.22, -40.55, -12.25) mm, rotated rx -180 ry 0 rz 90 deg; joints [72.744, -16.571, 81.712, 0, 24.858, 72.744]
  MoveL 7774 to (22.27, -39.5, -12.25) mm, rotated rx -180 ry 0 rz 90 deg; joints [72.767, -16.596, 81.804, 0, 24.791, 72.767]
  MoveL 7775 to (22.07, -39.33, -12.25) mm, rotated rx 180 ry 0 rz 90 deg; joints [72.771, -16.601, 81.823, 0, 24.778, 72.771]
  MoveL 7776 to (15.26, -33.64, -12.25) mm, rotated rx 180 ry 0 rz 90 deg; joints [72.884, -16.769, 82.442, 0, 24.327, 72.884]
  MoveL 7777 to (14.69, -33.17, -12.25) mm, rotated rx 180 ry 0 rz 90 deg; joints [72.893, -16.783, 82.493, 0, 24.29, 72.893]
  MoveL 7778 to (14.12, -32.69, -12.25) mm, rotated rx 180 ry 0 rz 90 deg; joints [72.903, -16.796, 82.544, 0, 24.252, 72.903]
  MoveC 7779 to (11.67, -32.23, -12.25) mm, rotated rx 180 ry 0 rz 90 deg; joints [72.894, -16.846, 82.731, 0, 24.116, 72.894] to (9.48, -33.43, -12.25) mm, rotated rx -180 ry 0 rz 90 deg; joints [72.834, -16.881, 82.861, 0, 24.02, 72.834]
  MoveL 7780 to (9.37, -33.64, -12.25) mm, rotated rx -180 ry 0 rz 90 deg; joints [72.826, -16.882, 82.864, 0, 24.018, 72.826]
  MoveL 7781 to (9.07, -34.59, -12.25) mm, rotated rx -180 ry 0 rz 90 deg; joints [72.793, -16.882, 82.865, 0, 24.018, 72.793]
  MoveL 7782 to (7.11, -41.72, -12.25) mm, rotated rx 180 ry 0 rz 90 deg; joints [72.547, -16.877, 82.846, 0, 24.031, 72.547]
  MoveL 7783 to (1.32, -63.02, -12.25) mm, rotated rx -180 ry 0 rz 90 deg; joints [71.813, -16.857, 82.77, 0, 24.087, 71.813]
  MoveL 7784 to (0.54, -65.86, -12.25) mm, rotated rx 180 ry 0 rz 90 deg; joints [71.715, -16.854, 82.759, 0, 24.095, 71.715]
  MoveL 7785 to (0.47, -66.1, -12.25) mm, rotated rx -180 ry 0 rz 90 deg; joints [71.707, -16.854, 82.758, 0, 24.096, 71.707]
  MoveL 7786 to (0.29, -66.81, -12.25) mm, rotated rx 180 ry 0 rz 90 deg; joints [71.683, -16.853, 82.754, 0, 24.098, 71.683]
  MoveC 7787 to (1.16, -69.24, -12.25) mm, rotated rx 180 ry 0 rz 90 deg; joints [71.615, -16.821, 82.635, 0, 24.186, 71.615] to (3.54, -70.21, -12.25) mm, rotated rx 180 ry 0 rz 90 deg; joints [71.609, -16.769, 82.442, 0, 24.327, 71.609]
  MoveC 7788 to (10.44, -69.98, -12.25) mm, rotated rx 180 ry 0 rz 90 deg; joints [71.689, -16.637, 81.954, 0, 24.683, 71.689] to (17.33, -69.7, -12.25) mm, rotated rx 180 ry 0 rz 90 deg; joints [71.769, -16.502, 81.463, 0, 25.039, 71.769]
  MoveL 7789 to (17, -62.16, -12.25) mm, rotated rx 180 ry 0 rz 90 deg; joints [72.002, -16.558, 81.665, 0, 24.892, 72.002]
  MoveL 7790 to (17, -62.16, -9.25) mm, rotated rx 180 ry 0 rz 90 deg; joints [72.002, -16.71, 81.768, 0, 24.942, 72.002]
  Establecer velocidad (1000.0 mm/s)
  MoveL 7791 to (17, -62.16, 10) mm, rotated rx 180 ry 0 rz 90 deg; joints [72.002, -17.684, 82.415, 0, 25.269, 72.002]
  Establecer velocidad (66.7 mm/s)
  MoveL 7792 to (22.4, 7.06, 10) mm, rotated rx 180 ry 0 rz 90 deg; joints [74.249, -17.994, 83.541, 0, 24.453, 74.249]
  MoveL 7793 to (22.4, 7.06, -9) mm, rotated rx 180 ry 0 rz 90 deg; joints [74.249, -17.028, 82.903, 0, 24.125, 74.249]
  MoveL 7794 to (23.89, 6.77, -9.41) mm, rotated rx 180 ry 0 rz 90 deg; joints [74.253, -16.977, 82.776, 0, 24.201, 74.253]
  MoveL 7795 to (25.41, 6.85, -9.81) mm, rotated rx -180 ry 0 rz 90 deg; joints [74.269, -16.927, 82.654, 0, 24.274, 74.269]
  MoveL 7796 to (26.87, 7.26, -10.22) mm, rotated rx -180 ry 0 rz 90 deg; joints [74.295, -16.881, 82.542, 0, 24.338, 74.295]
  MoveL 7797 to (28.21, 7.98, -10.62) mm, rotated rx 180 ry 0 rz 90 deg; joints [74.33, -16.838, 82.446, 0, 24.391, 74.33]
  MoveL 7798 to (29.35, 8.98, -11.03) mm, rotated rx -180 ry 0 rz 90 deg; joints [74.373, -16.8, 82.37, 0, 24.43, 74.373]
  MoveL 7799 to (30.24, 10.21, -11.44) mm, rotated rx 180 ry 0 rz 90 deg; joints [74.42, -16.769, 82.316, 0, 24.453, 74.42]
  MoveL 7800 to (30.84, 11.61, -11.84) mm, rotated rx -180 ry 0 rz 90 deg; joints [74.47, -16.744, 82.287, 0, 24.457, 74.47]
  MoveL 7801 to (31.09, 13.11, -12.25) mm, rotated rx 180 ry 0 rz 90 deg; joints [74.52, -16.727, 82.285, 0, 24.441, 74.52]
  MoveL 7802 to (31.1, 13.35, -12.25) mm, rotated rx -180 ry 0 rz 90 deg; joints [74.527, -16.728, 82.289, 0, 24.439, 74.527]
  MoveL 7803 to (31.1, 24.65, -12.25) mm, rotated rx 180 ry 0 rz 90 deg; joints [74.889, -16.788, 82.514, 0, 24.275, 74.889]
  MoveL 7804 to (16.58, 24.78, -12.25) mm, rotated rx 180 ry 0 rz 90 deg; joints [74.767, -17.067, 83.564, 0, 23.503, 74.767]
  MoveL 7805 to (15.49, 24.76, -12.25) mm, rotated rx 180 ry 0 rz 90 deg; joints [74.756, -17.088, 83.642, 0, 23.446, 74.756]
  MoveC 7806 to (13.19, 23.71, -12.25) mm, rotated rx 180 ry 0 rz 90 deg; joints [74.702, -17.126, 83.787, 0, 23.339, 74.702] to (12.37, 21.32, -12.25) mm, rotated rx 180 ry 0 rz 90 deg; joints [74.618, -17.129, 83.798, 0, 23.331, 74.618]
  MoveL 7807 to (12.52, 20.85, -12.25) mm, rotated rx -180 ry 0 rz 90 deg; joints [74.604, -17.124, 83.778, 0, 23.345, 74.604]
  MoveL 7808 to (15.64, 12.46, -12.25) mm, rotated rx 180 ry 0 rz 90 deg; joints [74.361, -17.021, 83.388, 0, 23.633, 74.361]
  MoveL 7809 to (15.9, 11.8, -12.25) mm, rotated rx -180 ry 0 rz 90 deg; joints [74.342, -17.013, 83.356, 0, 23.657, 74.342]
  MoveC 7810 to (16.2, 11.25, -12.25) mm, rotated rx -180 ry 0 rz 90 deg; joints [74.327, -17.004, 83.323, 0, 23.681, 74.327] to (16.65, 10.8, -12.25) mm, rotated rx -180 ry 0 rz 90 deg; joints [74.317, -16.993, 83.282, 0, 23.711, 74.317]
  MoveL 7811 to (17.53, 10.12, -12.25) mm, rotated rx 180 ry 0 rz 90 deg; joints [74.303, -16.973, 83.205, 0, 23.768, 74.303]
  MoveL 7812 to (27.96, 2.5, -12.25) mm, rotated rx 180 ry 0 rz 90 deg; joints [74.153, -16.73, 82.297, 0, 24.433, 74.153]
  MoveL 7813 to (28.34, 2.24, -12.25) mm, rotated rx 180 ry 0 rz 90 deg; joints [74.148, -16.721, 82.264, 0, 24.457, 74.148]
  MoveC 7814 to (29.69, 1.76, -12.25) mm, rotated rx 180 ry 0 rz 90 deg; joints [74.145, -16.691, 82.155, 0, 24.536, 74.145] to (31.1, 2.04, -12.25) mm, rotated rx 180 ry 0 rz 90 deg; joints [74.167, -16.665, 82.058, 0, 24.607, 74.167]
